// TIA Portal project "tiaS7libCommunication" (V15)

(* hardware
DEVICE "S7-1200 station_1"  S7-1200 Station
   slot 0: "Rack_0"  S7-1200 Rack  Rack  V1.0
   slot 1: "PLC_1"  CPU 1214C DC/DC/DC  6ES7 214-1AG40-0XB0  V4.2
DEVICE "HMI_1"  KTP700 Basic PN
   slot 0: "HMI_1"  KTP700 Basic PN  6AV2 123-2GB03-0AX0  15.0.0.0
   slot 1: "HMI_RT_1"  KTP700 Basic PN  6AV2 123-2GB03-0AX0  15.0.0.0
   slot 5: "HMI_1.IE_CP_1"  PROFINET Interface  15.0.0.0
      slot 1: "PROFINET Interface_1"  PROFINET Interface
         slot 1: "Port_1"  Port
DEVICE "HMI_2"  TP1500 Comfort
   slot 0: "HMI_2"  TP1500 Comfort  6AV2 124-0QC02-0AX1  15.0.0.0
   slot 1: "HMI_RT_2"  TP1500 Comfort  6AV2 124-0QC02-0AX1  15.0.0.0
   slot 5: "HMI_2.IE_CP_1"  PROFINET Interface  15.0.0.0
      slot 1: "PROFINET Interface_1"  PROFINET Interface
         slot 1: "Port_1"  Port
         slot 2: "Port_2"  Port
   slot 6: "HMI_2.IE_CP_2"  PROFINET Interface  15.0.0.0
      slot 1: "PROFINET Interface_GBit"  PROFINET Interface
         slot 1: "Port_1"  Port
   slot 7: "HMI_2.MPI/DP_CP_1"  MPI/DP Interface  15.0.0.0
*)

// ===== PLC "PLC_1"  CPU 1214C DC/DC/DC =====

VAR_GLOBAL   // PLC tag table "Default tag table"
   "o_test_valve_start" AT %M0.0 : Bool;
   "o_test_valve_end" AT %M0.1 : Bool;
   "i_test_valve_start" AT %M0.2 : Bool;
   "i_test_vavlve_end" AT %M0.3 : Bool;
END_VAR

TYPE "TestSuite"
   STRUCT
      tc_name : Array[1..64] of String[127];
      tc_size : Byte;
      ts_name : String[127];
   END_STRUCT;
END_TYPE

TYPE "UnitLib"
   STRUCT
      "step" : Int;
      input_buffer : Array[0..3] of Byte;
      output_buffer : Array[0..127] of Byte;
      output_len : UDInt;
      network_id : Conn_Ouc := 1;
      unit : Array[1..3] of "TestSuite";
      ts_size : Byte := 3;
   END_STRUCT;
   // unit[1].tc_size := 8;
   // unit[2].tc_name[2] := 'cb_insert_glass_test';
   // unit[2].tc_name[1] := 'cb_get_glass_info_test';
   // unit[1].ts_name := 'Priority queue test';
   // unit[2].tc_size := 16#7;
   // unit[1].tc_name[1] := 'pq_enqueue_test';
   // unit[1].tc_name[2] := 'pq_size_test';
   // unit[1].tc_name[3] := 'pq_is_empty_test';
   // unit[1].tc_name[8] := 'pq_clear_test';
   // unit[1].tc_name[4] := 'pq_peek_test';
   // unit[1].tc_name[5] := 'pq_delete_by_index_test';
   // unit[1].tc_name[6] := 'pq_dequeue_test';
   // unit[1].tc_name[7] := 'pq_find_by_vehicle_number_test';
   // unit[2].ts_name := 'Curing buffer test';
   // unit[2].tc_name[3] := 'cb_is_drawer_enabled_test';
   // unit[2].tc_name[4] := 'cb_is_drawer_free_test';
   // unit[2].tc_name[5] := 'cb_is_glass_expired_test';
   // unit[2].tc_name[7] := 'cb_remove_glass_test';
   // unit[2].tc_name[6] := 'cb_is_glass_ready_test';
   // unit[3].ts_name := 'Centering bed test';
   // unit[3].tc_name[1] := 'centering_bed_do_centering_test';
   // unit[3].tc_name[2] := 'centering_bed_get_state_test';
   // unit[3].tc_name[3] := 'centering_bed_is_centered_test';
   // unit[3].tc_name[4] := 'centering_bed_is_occupied_test';
   // unit[3].tc_name[5] := 'centering_bed_release_centering_test';
   // unit[3].tc_size := 16#5;
END_TYPE

TYPE "GlassInfo"
   STRUCT
      vehicle_number : String[100];
      vehicle_model : String[50];
      rear_window : String[50];
   END_STRUCT;
END_TYPE

TYPE "Valve2Pos"
   STRUCT
      status_error : Bool;   // error status, valve not reacts
      cmd_end_position : Bool;   // state conditional variable for setting valve end position
      cmd_start_position : Bool;   // state conditional variable for setting valve start position
      request_signal_start : Bool;   // request for set valve to start position
      request_signal_end : Bool;   // request for set valve to end position
      request_release : Bool;   // request for release valve (no output signals)
      watchdog_timer : TON_TIME;   // timer for reaction of valve
      reaction_delay : Time;   // delay for reaction of valve
      io : "IOValve2pos";
   END_STRUCT;
END_TYPE

// folder: CenteringBed

TYPE "CenteringBed"
   STRUCT
      "step" : Int;
      manual_mode_interface : "CenteringBedManual";
      x_centering_valve : "Valve2Pos";
      y_centering_valve : "Valve2Pos";
      suction_cup_lifting_cylinder : "Valve2Pos";
      status_error : Bool;
      cmd_vacuum : Bool;
      request_reset_error : Bool;
      io : "IOCenterngBed";
   END_STRUCT;
END_TYPE

TYPE "CenteringBedManual"
   STRUCT
      manual_mode : Bool;
      manual_anutomat_mode : Bool;
      request_manual_centering_x : Bool;
      request_manual_centering_y : Bool;
      request_manual_cuction_cup_lifting : Bool;
      request_manual_vacuum : Bool;
      request_manual_eject : Bool;
      request_do_manual_centering : Bool;
      request_manual_release_centering : Bool;
   END_STRUCT;
END_TYPE

// folder: CuringBuffer

TYPE "CuringBuffer"
   STRUCT
      drawer_array : Array[0..7] of "CuringBufferDrawer";
      min_expiration_time : Time;
      max_expiration_time : Time;
      drawer_count : Int := 8;
   END_STRUCT;
END_TYPE

TYPE "CuringBufferDrawer"
   STRUCT
      enable : Bool;
      occupied : Bool;
      presence_sensor : Bool;
      insertion_time : DTL;
      glass : "GlassInfo";
   END_STRUCT;
END_TYPE

// folder: MES

TYPE "MesPlcParams"
   STRUCT
      InitialPLC : Bool;   // InitialPLC
      InitialServerAck : Bool;   // InitialServerAck
      CycleRequest : Bool;   // CycleRequest
      CycleSuccess : Bool;   // CycleSuccess
      CycleFailure : Bool;   // CycleFailure
      CycleAbort : Bool;   // CycleAbort
      RES_501 : Byte;   // Reserviert
      RES_502 : Byte;   // Reserviert
      RES_503 : Byte;   // Reserviert
      PartSerialPLC : Array[1..40] of Char;   // PartSerialPLC
      ProcessDataCount : Int;   // ProcessDataCount <n>
      RES_546 : Array[0..126] of Word;   // Reserviert
      KeyProcessData : Array[1..50] of Char;   // Für jeden Index <i> von 0 bis <n> -1
      ValueProcessData : Array[1..50] of Char;   // Für jeden Index <i> von 0 bis <n> -1
   END_STRUCT;
   // PartSerialPLC[1] := '$00';
   // PartSerialPLC[2] := '$00';
   // PartSerialPLC[3] := '$00';
   // PartSerialPLC[4] := '$00';
   // PartSerialPLC[5] := '$00';
   // PartSerialPLC[6] := '$00';
   // PartSerialPLC[7] := '$00';
   // PartSerialPLC[8] := '$00';
   // PartSerialPLC[9] := '$00';
   // PartSerialPLC[10] := '$00';
   // PartSerialPLC[11] := '$00';
   // PartSerialPLC[12] := '$00';
   // PartSerialPLC[13] := '$00';
   // PartSerialPLC[14] := '$00';
   // PartSerialPLC[15] := '$00';
   // PartSerialPLC[16] := '$00';
   // PartSerialPLC[17] := '$00';
   // PartSerialPLC[18] := '$00';
   // PartSerialPLC[19] := '$00';
   // PartSerialPLC[20] := '$00';
   // PartSerialPLC[21] := '$00';
   // PartSerialPLC[22] := '$00';
   // PartSerialPLC[23] := '$00';
   // PartSerialPLC[24] := '$00';
   // PartSerialPLC[25] := '$00';
   // PartSerialPLC[26] := '$00';
   // PartSerialPLC[27] := '$00';
   // PartSerialPLC[28] := '$00';
   // PartSerialPLC[29] := '$00';
   // PartSerialPLC[30] := '$00';
   // PartSerialPLC[31] := '$00';
   // PartSerialPLC[32] := '$00';
   // PartSerialPLC[33] := '$00';
   // PartSerialPLC[34] := '$00';
   // PartSerialPLC[35] := '$00';
   // PartSerialPLC[36] := '$00';
   // PartSerialPLC[37] := '$00';
   // PartSerialPLC[38] := '$00';
   // PartSerialPLC[39] := '$00';
   // PartSerialPLC[40] := '$00';
   // KeyProcessData[1] := '$00';
   // KeyProcessData[2] := '$00';
   // KeyProcessData[3] := '$00';
   // KeyProcessData[4] := '$00';
   // KeyProcessData[5] := '$00';
   // KeyProcessData[6] := '$00';
   // KeyProcessData[7] := '$00';
   // KeyProcessData[8] := '$00';
   // KeyProcessData[9] := '$00';
   // KeyProcessData[10] := '$00';
   // KeyProcessData[11] := '$00';
   // KeyProcessData[12] := '$00';
   // KeyProcessData[13] := '$00';
   // KeyProcessData[14] := '$00';
   // KeyProcessData[15] := '$00';
   // KeyProcessData[16] := '$00';
   // KeyProcessData[17] := '$00';
   // KeyProcessData[18] := '$00';
   // KeyProcessData[19] := '$00';
   // KeyProcessData[20] := '$00';
   // KeyProcessData[21] := '$00';
   // KeyProcessData[22] := '$00';
   // KeyProcessData[23] := '$00';
   // KeyProcessData[24] := '$00';
   // KeyProcessData[25] := '$00';
   // KeyProcessData[26] := '$00';
   // KeyProcessData[27] := '$00';
   // KeyProcessData[28] := '$00';
   // KeyProcessData[29] := '$00';
   // KeyProcessData[30] := '$00';
   // KeyProcessData[31] := '$00';
   // KeyProcessData[32] := '$00';
   // KeyProcessData[33] := '$00';
   // KeyProcessData[34] := '$00';
   // KeyProcessData[35] := '$00';
   // KeyProcessData[36] := '$00';
   // KeyProcessData[37] := '$00';
   // KeyProcessData[38] := '$00';
   // KeyProcessData[39] := '$00';
   // KeyProcessData[40] := '$00';
   // KeyProcessData[41] := '$00';
   // KeyProcessData[42] := '$00';
   // KeyProcessData[43] := '$00';
   // KeyProcessData[44] := '$00';
   // KeyProcessData[45] := '$00';
   // KeyProcessData[46] := '$00';
   // KeyProcessData[47] := '$00';
   // KeyProcessData[48] := '$00';
   // KeyProcessData[49] := '$00';
   // KeyProcessData[50] := '$00';
   // ValueProcessData[1] := '$00';
   // ValueProcessData[2] := '$00';
   // ValueProcessData[3] := '$00';
   // ValueProcessData[4] := '$00';
   // ValueProcessData[5] := '$00';
   // ValueProcessData[6] := '$00';
   // ValueProcessData[7] := '$00';
   // ValueProcessData[8] := '$00';
   // ValueProcessData[9] := '$00';
   // ValueProcessData[10] := '$00';
   // ValueProcessData[11] := '$00';
   // ValueProcessData[12] := '$00';
   // ValueProcessData[13] := '$00';
   // ValueProcessData[14] := '$00';
   // ValueProcessData[15] := '$00';
   // ValueProcessData[16] := '$00';
   // ValueProcessData[17] := '$00';
   // ValueProcessData[18] := '$00';
   // ValueProcessData[19] := '$00';
   // ValueProcessData[20] := '$00';
   // ValueProcessData[21] := '$00';
   // ValueProcessData[22] := '$00';
   // ValueProcessData[23] := '$00';
   // ValueProcessData[24] := '$00';
   // ValueProcessData[25] := '$00';
   // ValueProcessData[26] := '$00';
   // ValueProcessData[27] := '$00';
   // ValueProcessData[28] := '$00';
   // ValueProcessData[29] := '$00';
   // ValueProcessData[30] := '$00';
   // ValueProcessData[31] := '$00';
   // ValueProcessData[32] := '$00';
   // ValueProcessData[33] := '$00';
   // ValueProcessData[34] := '$00';
   // ValueProcessData[35] := '$00';
   // ValueProcessData[36] := '$00';
   // ValueProcessData[37] := '$00';
   // ValueProcessData[38] := '$00';
   // ValueProcessData[39] := '$00';
   // ValueProcessData[40] := '$00';
   // ValueProcessData[41] := '$00';
   // ValueProcessData[42] := '$00';
   // ValueProcessData[43] := '$00';
   // ValueProcessData[44] := '$00';
   // ValueProcessData[45] := '$00';
   // ValueProcessData[46] := '$00';
   // ValueProcessData[47] := '$00';
   // ValueProcessData[48] := '$00';
   // ValueProcessData[49] := '$00';
   // ValueProcessData[50] := '$00';
END_TYPE

TYPE "MesServerParams"
   STRUCT
      LiveCheck : Bool;   // LiveCheck, vom Server gesetzt
      RES_001 : Byte;   // Reserviert
      InitialServer : Bool;   // InitialServer
      InitialPLCAck : Bool;   // InitialPLCAck
      ReadyForCycle : Bool;   // ReadyForCycle
      CycleRequestAck : Bool;   // CycleRequestAck
      CycleRequestReject : Bool;   // CycleRequestReject
      CycleAck : Bool;   // CycleAck
      RES_003 : Byte;   // Reserviert
      PartSerial : Array[1..40] of Char;   // PartSerial
      ParameterBarcode : Array[1..100] of Char;   // ParameterBarcode
      Error_Reason_Code : Int;
      ErrorMessage : Array[1..200] of Char;   // ErrorMessage
      Reserve : Array[1..154] of Char;   // Reserve
   END_STRUCT;
   // PartSerial[1] := '$00';
   // PartSerial[2] := '$00';
   // PartSerial[3] := '$00';
   // PartSerial[4] := '$00';
   // PartSerial[5] := '$00';
   // PartSerial[6] := '$00';
   // PartSerial[7] := '$00';
   // PartSerial[8] := '$00';
   // PartSerial[9] := '$00';
   // PartSerial[10] := '$00';
   // PartSerial[11] := '$00';
   // PartSerial[12] := '$00';
   // PartSerial[13] := '$00';
   // PartSerial[14] := '$00';
   // PartSerial[15] := '$00';
   // PartSerial[16] := '$00';
   // PartSerial[17] := '$00';
   // PartSerial[18] := '$00';
   // PartSerial[19] := '$00';
   // PartSerial[20] := '$00';
   // PartSerial[21] := '$00';
   // PartSerial[22] := '$00';
   // PartSerial[23] := '$00';
   // PartSerial[24] := '$00';
   // PartSerial[25] := '$00';
   // PartSerial[26] := '$00';
   // PartSerial[27] := '$00';
   // PartSerial[28] := '$00';
   // PartSerial[29] := '$00';
   // PartSerial[30] := '$00';
   // PartSerial[31] := '$00';
   // PartSerial[32] := '$00';
   // PartSerial[33] := '$00';
   // PartSerial[34] := '$00';
   // PartSerial[35] := '$00';
   // PartSerial[36] := '$00';
   // PartSerial[37] := '$00';
   // PartSerial[38] := '$00';
   // PartSerial[39] := '$00';
   // PartSerial[40] := '$00';
   // ParameterBarcode[1] := '$00';
   // ParameterBarcode[2] := '$00';
   // ParameterBarcode[3] := '$00';
   // ParameterBarcode[4] := '$00';
   // ParameterBarcode[5] := '$00';
   // ParameterBarcode[6] := '$00';
   // ParameterBarcode[7] := '$00';
   // ParameterBarcode[8] := '$00';
   // ParameterBarcode[9] := '$00';
   // ParameterBarcode[10] := '$00';
   // ParameterBarcode[11] := '$00';
   // ParameterBarcode[12] := '$00';
   // ParameterBarcode[13] := '$00';
   // ParameterBarcode[14] := '$00';
   // ParameterBarcode[15] := '$00';
   // ParameterBarcode[16] := '$00';
   // ParameterBarcode[17] := '$00';
   // ParameterBarcode[18] := '$00';
   // ParameterBarcode[19] := '$00';
   // ParameterBarcode[20] := '$00';
   // ParameterBarcode[21] := '$00';
   // ParameterBarcode[22] := '$00';
   // ParameterBarcode[23] := '$00';
   // ParameterBarcode[24] := '$00';
   // ParameterBarcode[25] := '$00';
   // ParameterBarcode[26] := '$00';
   // ParameterBarcode[27] := '$00';
   // ParameterBarcode[28] := '$00';
   // ParameterBarcode[29] := '$00';
   // ParameterBarcode[30] := '$00';
   // ParameterBarcode[31] := '$00';
   // ParameterBarcode[32] := '$00';
   // ParameterBarcode[33] := '$00';
   // ParameterBarcode[34] := '$00';
   // ParameterBarcode[35] := '$00';
   // ParameterBarcode[36] := '$00';
   // ParameterBarcode[37] := '$00';
   // ParameterBarcode[38] := '$00';
   // ParameterBarcode[39] := '$00';
   // ParameterBarcode[40] := '$00';
   // ParameterBarcode[41] := '$00';
   // ParameterBarcode[42] := '$00';
   // ParameterBarcode[43] := '$00';
   // ParameterBarcode[44] := '$00';
   // ParameterBarcode[45] := '$00';
   // ParameterBarcode[46] := '$00';
   // ParameterBarcode[47] := '$00';
   // ParameterBarcode[48] := '$00';
   // ParameterBarcode[49] := '$00';
   // ParameterBarcode[50] := '$00';
   // ParameterBarcode[51] := '$00';
   // ParameterBarcode[52] := '$00';
   // ParameterBarcode[53] := '$00';
   // ParameterBarcode[54] := '$00';
   // ParameterBarcode[55] := '$00';
   // ParameterBarcode[56] := '$00';
   // ParameterBarcode[57] := '$00';
   // ParameterBarcode[58] := '$00';
   // ParameterBarcode[59] := '$00';
   // ParameterBarcode[60] := '$00';
   // ParameterBarcode[61] := '$00';
   // ParameterBarcode[62] := '$00';
   // ParameterBarcode[63] := '$00';
   // ParameterBarcode[64] := '$00';
   // ParameterBarcode[65] := '$00';
   // ParameterBarcode[66] := '$00';
   // ParameterBarcode[67] := '$00';
   // ParameterBarcode[68] := '$00';
   // ParameterBarcode[69] := '$00';
   // ParameterBarcode[70] := '$00';
   // ParameterBarcode[71] := '$00';
   // ParameterBarcode[72] := '$00';
   // ParameterBarcode[73] := '$00';
   // ParameterBarcode[74] := '$00';
   // ParameterBarcode[75] := '$00';
   // ParameterBarcode[76] := '$00';
   // ParameterBarcode[77] := '$00';
   // ParameterBarcode[78] := '$00';
   // ParameterBarcode[79] := '$00';
   // ParameterBarcode[80] := '$00';
   // ParameterBarcode[81] := '$00';
   // ParameterBarcode[82] := '$00';
   // ParameterBarcode[83] := '$00';
   // ParameterBarcode[84] := '$00';
   // ParameterBarcode[85] := '$00';
   // ParameterBarcode[86] := '$00';
   // ParameterBarcode[87] := '$00';
   // ParameterBarcode[88] := '$00';
   // ParameterBarcode[89] := '$00';
   // ParameterBarcode[90] := '$00';
   // ParameterBarcode[91] := '$00';
   // ParameterBarcode[92] := '$00';
   // ParameterBarcode[93] := '$00';
   // ParameterBarcode[94] := '$00';
   // ParameterBarcode[95] := '$00';
   // ParameterBarcode[96] := '$00';
   // ParameterBarcode[97] := '$00';
   // ParameterBarcode[98] := '$00';
   // ParameterBarcode[99] := '$00';
   // ParameterBarcode[100] := '$00';
END_TYPE

// folder: PriorityQueue

TYPE "PriorityQueue"
   STRUCT
      array_size : Int := 100;
      size : Int;
      queue_array : Array[0..99] of "QueueNode";
   END_STRUCT;
END_TYPE

TYPE "QueueNode"
   STRUCT
      allocated : Bool;
      priority : Bool;
      glass : "GlassInfo";
   END_STRUCT;
END_TYPE

// folder: Queue

TYPE "queue_pc"
   STRUCT
      visual_queue : Array[0..9] of "GlassInfo";
      cmd_done : Bool;
   END_STRUCT;
END_TYPE

TYPE "queue_plc"
   STRUCT
      glass : "GlassInfo";
      cmd_add : Bool;
      cmd_add_priority : Bool;
      cmd_delete : Bool;
   END_STRUCT;
END_TYPE

// folder: io

TYPE "IOCuringBuffer"
   STRUCT
      presence_sensor_drawer_0 : Bool;
      presence_sensor_drawer_1 : Bool;
      presence_sensor_drawer_2 : Bool;
      presence_sensor_drawer_3 : Bool;
      presence_sensor_drawer_4 : Bool;
      presence_sensor_drawer_5 : Bool;
      presence_sensor_drawer_6 : Bool;
      presence_sensor_drawer_7 : Bool;
   END_STRUCT;
END_TYPE

TYPE "IOCenterngBed"
   STRUCT
      i_vacuum : Bool;
      i_glass_presence_sensor : Bool;
      o_vacuum : Bool;
      o_eject : Bool;
      centering_x_valve_io : "IOValve2pos";
      centering_y_valve_io : "IOValve2pos";
      suction_cup_lifting_io : "IOValve2pos";
   END_STRUCT;
END_TYPE

TYPE "IOValve2pos"
   STRUCT
      i_start_position : Bool;
      i_end_position : Bool;
      o_start_position : Bool;
      o_end_position : Bool;
   END_STRUCT;
END_TYPE

// folder: (top level)

DATA_BLOCK "PLCUnitLib_DB"   // DB2
{ S7_Optimized_Access := 'TRUE' }
VERSION : 0.1
// stored: InstanceOfName PLCUnitLib
"PLCUnitLib"
BEGIN
END_DATA_BLOCK

DATA_BLOCK "Valves_DB"   // DB3
{ S7_Optimized_Access := 'TRUE' }
VERSION : 0.1
   VAR
      test_valve : "Valve2Pos";
   END_VAR
BEGIN
END_DATA_BLOCK

DATA_BLOCK "io_sync_DB"   // DB4
{ S7_Optimized_Access := 'TRUE' }
VERSION : 0.1
// stored: InstanceOfName io_sync
"io_sync"
BEGIN
END_DATA_BLOCK

DATA_BLOCK "db_queue"   // DB5
{ S7_Optimized_Access := 'FALSE' }
VERSION : 0.1
   VAR
      plc : "queue_plc";
      pc : "queue_pc";
   END_VAR
BEGIN
   plc.glass.vehicle_number := '123456789 00';
   plc.glass.vehicle_model := 'IDBuzz';
   plc.glass.rear_window := 'VW-Number';
END_DATA_BLOCK

DATA_BLOCK "DB_MES_V2"   // DB6
{ S7_Optimized_Access := 'FALSE' }
VERSION : 0.1
   VAR
      MES : "MesServerParams";
      PLC : "MesPlcParams";
   END_VAR
BEGIN
END_DATA_BLOCK

DATA_BLOCK "DB_process_data"   // DB7
{ S7_Optimized_Access := 'TRUE' }
VERSION : 0.1
   VAR
      glass_queue : "PriorityQueue";
   END_VAR
   VAR RETAIN
      curing_buffer_1 : "CuringBuffer";
   END_VAR
   VAR
      centering_bed : "CenteringBed";
   END_VAR
BEGIN
END_DATA_BLOCK

DATA_BLOCK "DB_MES"   // DB600
{ S7_Optimized_Access := 'FALSE' }
VERSION : 0.1
   VAR
      LiveCheck : Bool;   // LiveCheck, vom Server gesetzt
      RES_001 : Byte;   // Reserviert
      InitialServer : Bool;   // InitialServer
      InitialPLCAck : Bool;   // InitialPLCAck
      ReadyForCycle : Bool;   // ReadyForCycle
      CycleRequestAck : Bool;   // CycleRequestAck
      CycleRequestReject : Bool;   // CycleRequestReject
      CycleAck : Bool;   // CycleAck
      RES_003 : Byte;   // Reserviert
      PartSerial : Array[1..40] of Char;   // PartSerial
      ParameterBarcode : Array[1..100] of Char;   // ParameterBarcode
      Error_Reason_Code : Int;
      ErrorMessage : Array[1..200] of Char;   // ErrorMessage
      Reserve : Array[1..154] of Char;   // Reserve
      InitialPLC : Bool;   // InitialPLC
      InitialServerAck : Bool;   // InitialServerAck
      CycleRequest : Bool;   // CycleRequest
      CycleSuccess : Bool;   // CycleSuccess
      CycleFailure : Bool;   // CycleFailure
      CycleAbort : Bool;   // CycleAbort
      RES_501 : Byte;   // Reserviert
      RES_502 : Byte;   // Reserviert
      RES_503 : Byte;   // Reserviert
      PartSerialPLC : Array[1..40] of Char;   // PartSerialPLC
      ProcessDataCount : Int;   // ProcessDataCount <n>
      RES_546 : Array[0..126] of Word;   // Reserviert
      KeyProcessData : Array[1..50] of Char;   // Für jeden Index <i> von 0 bis <n> -1
      ValueProcessData : Array[1..50] of Char;   // Für jeden Index <i> von 0 bis <n> -1
   END_VAR
BEGIN
   ValueProcessData[50] := '$00';
   ValueProcessData[1] := '$00';
   ValueProcessData[2] := '$00';
   ValueProcessData[3] := '$00';
   ValueProcessData[4] := '$00';
   ValueProcessData[5] := '$00';
   ValueProcessData[6] := '$00';
   ValueProcessData[7] := '$00';
   ValueProcessData[8] := '$00';
   ValueProcessData[9] := '$00';
   ValueProcessData[10] := '$00';
   ValueProcessData[11] := '$00';
   ValueProcessData[12] := '$00';
   ValueProcessData[13] := '$00';
   ValueProcessData[14] := '$00';
   ValueProcessData[15] := '$00';
   ValueProcessData[16] := '$00';
   ValueProcessData[17] := '$00';
   ValueProcessData[18] := '$00';
   ValueProcessData[19] := '$00';
   ValueProcessData[20] := '$00';
   ValueProcessData[21] := '$00';
   ValueProcessData[22] := '$00';
   ValueProcessData[23] := '$00';
   ValueProcessData[24] := '$00';
   ValueProcessData[25] := '$00';
   ValueProcessData[26] := '$00';
   ValueProcessData[27] := '$00';
   ValueProcessData[28] := '$00';
   ValueProcessData[29] := '$00';
   ValueProcessData[30] := '$00';
   ValueProcessData[31] := '$00';
   ValueProcessData[32] := '$00';
   ValueProcessData[33] := '$00';
   ValueProcessData[34] := '$00';
   ValueProcessData[35] := '$00';
   ValueProcessData[36] := '$00';
   ValueProcessData[37] := '$00';
   ValueProcessData[38] := '$00';
   ValueProcessData[39] := '$00';
   ValueProcessData[40] := '$00';
   ValueProcessData[41] := '$00';
   ValueProcessData[42] := '$00';
   ValueProcessData[43] := '$00';
   ValueProcessData[44] := '$00';
   ValueProcessData[45] := '$00';
   ValueProcessData[46] := '$00';
   ValueProcessData[47] := '$00';
   ValueProcessData[48] := '$00';
   ValueProcessData[49] := '$00';
   KeyProcessData[1] := '$00';
   KeyProcessData[2] := '$00';
   KeyProcessData[3] := '$00';
   KeyProcessData[4] := '$00';
   KeyProcessData[5] := '$00';
   KeyProcessData[6] := '$00';
   KeyProcessData[7] := '$00';
   KeyProcessData[8] := '$00';
   KeyProcessData[9] := '$00';
   KeyProcessData[10] := '$00';
   KeyProcessData[11] := '$00';
   KeyProcessData[12] := '$00';
   KeyProcessData[13] := '$00';
   KeyProcessData[14] := '$00';
   KeyProcessData[15] := '$00';
   KeyProcessData[16] := '$00';
   KeyProcessData[17] := '$00';
   KeyProcessData[18] := '$00';
   KeyProcessData[19] := '$00';
   KeyProcessData[20] := '$00';
   KeyProcessData[21] := '$00';
   KeyProcessData[22] := '$00';
   KeyProcessData[23] := '$00';
   KeyProcessData[24] := '$00';
   KeyProcessData[25] := '$00';
   KeyProcessData[26] := '$00';
   KeyProcessData[27] := '$00';
   KeyProcessData[28] := '$00';
   KeyProcessData[29] := '$00';
   KeyProcessData[30] := '$00';
   KeyProcessData[31] := '$00';
   KeyProcessData[32] := '$00';
   KeyProcessData[33] := '$00';
   KeyProcessData[34] := '$00';
   KeyProcessData[35] := '$00';
   KeyProcessData[36] := '$00';
   KeyProcessData[37] := '$00';
   KeyProcessData[38] := '$00';
   KeyProcessData[39] := '$00';
   KeyProcessData[40] := '$00';
   KeyProcessData[41] := '$00';
   KeyProcessData[42] := '$00';
   KeyProcessData[43] := '$00';
   KeyProcessData[44] := '$00';
   KeyProcessData[45] := '$00';
   KeyProcessData[46] := '$00';
   KeyProcessData[47] := '$00';
   KeyProcessData[48] := '$00';
   KeyProcessData[49] := '$00';
   KeyProcessData[50] := '$00';
   PartSerialPLC[1] := '$00';
   PartSerialPLC[2] := '$00';
   PartSerialPLC[3] := '$00';
   PartSerialPLC[4] := '$00';
   PartSerialPLC[5] := '$00';
   PartSerialPLC[6] := '$00';
   PartSerialPLC[7] := '$00';
   PartSerialPLC[8] := '$00';
   PartSerialPLC[9] := '$00';
   PartSerialPLC[10] := '$00';
   PartSerialPLC[11] := '$00';
   PartSerialPLC[12] := '$00';
   PartSerialPLC[13] := '$00';
   PartSerialPLC[14] := '$00';
   PartSerialPLC[15] := '$00';
   PartSerialPLC[16] := '$00';
   PartSerialPLC[17] := '$00';
   PartSerialPLC[18] := '$00';
   PartSerialPLC[19] := '$00';
   PartSerialPLC[20] := '$00';
   PartSerialPLC[21] := '$00';
   PartSerialPLC[22] := '$00';
   PartSerialPLC[23] := '$00';
   PartSerialPLC[24] := '$00';
   PartSerialPLC[25] := '$00';
   PartSerialPLC[26] := '$00';
   PartSerialPLC[27] := '$00';
   PartSerialPLC[28] := '$00';
   PartSerialPLC[29] := '$00';
   PartSerialPLC[30] := '$00';
   PartSerialPLC[31] := '$00';
   PartSerialPLC[32] := '$00';
   PartSerialPLC[33] := '$00';
   PartSerialPLC[34] := '$00';
   PartSerialPLC[35] := '$00';
   PartSerialPLC[36] := '$00';
   PartSerialPLC[37] := '$00';
   PartSerialPLC[38] := '$00';
   PartSerialPLC[39] := '$00';
   PartSerialPLC[40] := '$00';
   PartSerial[1] := '$00';
   PartSerial[2] := '$00';
   PartSerial[3] := '$00';
   PartSerial[4] := '$00';
   PartSerial[5] := '$00';
   PartSerial[6] := '$00';
   PartSerial[7] := '$00';
   PartSerial[8] := '$00';
   PartSerial[9] := '$00';
   PartSerial[10] := '$00';
   PartSerial[11] := '$00';
   PartSerial[12] := '$00';
   PartSerial[13] := '$00';
   PartSerial[14] := '$00';
   PartSerial[15] := '$00';
   PartSerial[16] := '$00';
   PartSerial[17] := '$00';
   PartSerial[18] := '$00';
   PartSerial[19] := '$00';
   PartSerial[20] := '$00';
   PartSerial[21] := '$00';
   PartSerial[22] := '$00';
   PartSerial[23] := '$00';
   PartSerial[24] := '$00';
   PartSerial[25] := '$00';
   PartSerial[26] := '$00';
   PartSerial[27] := '$00';
   PartSerial[28] := '$00';
   PartSerial[29] := '$00';
   PartSerial[30] := '$00';
   PartSerial[31] := '$00';
   PartSerial[32] := '$00';
   PartSerial[33] := '$00';
   PartSerial[34] := '$00';
   PartSerial[35] := '$00';
   PartSerial[36] := '$00';
   PartSerial[37] := '$00';
   PartSerial[38] := '$00';
   PartSerial[39] := '$00';
   PartSerial[40] := '$00';
   ParameterBarcode[1] := '$00';
   ParameterBarcode[2] := '$00';
   ParameterBarcode[3] := '$00';
   ParameterBarcode[4] := '$00';
   ParameterBarcode[5] := '$00';
   ParameterBarcode[6] := '$00';
   ParameterBarcode[7] := '$00';
   ParameterBarcode[8] := '$00';
   ParameterBarcode[9] := '$00';
   ParameterBarcode[10] := '$00';
   ParameterBarcode[11] := '$00';
   ParameterBarcode[12] := '$00';
   ParameterBarcode[13] := '$00';
   ParameterBarcode[14] := '$00';
   ParameterBarcode[15] := '$00';
   ParameterBarcode[16] := '$00';
   ParameterBarcode[17] := '$00';
   ParameterBarcode[18] := '$00';
   ParameterBarcode[19] := '$00';
   ParameterBarcode[20] := '$00';
   ParameterBarcode[21] := '$00';
   ParameterBarcode[22] := '$00';
   ParameterBarcode[23] := '$00';
   ParameterBarcode[24] := '$00';
   ParameterBarcode[25] := '$00';
   ParameterBarcode[26] := '$00';
   ParameterBarcode[27] := '$00';
   ParameterBarcode[28] := '$00';
   ParameterBarcode[29] := '$00';
   ParameterBarcode[30] := '$00';
   ParameterBarcode[31] := '$00';
   ParameterBarcode[32] := '$00';
   ParameterBarcode[33] := '$00';
   ParameterBarcode[34] := '$00';
   ParameterBarcode[35] := '$00';
   ParameterBarcode[36] := '$00';
   ParameterBarcode[37] := '$00';
   ParameterBarcode[38] := '$00';
   ParameterBarcode[39] := '$00';
   ParameterBarcode[40] := '$00';
   ParameterBarcode[41] := '$00';
   ParameterBarcode[42] := '$00';
   ParameterBarcode[43] := '$00';
   ParameterBarcode[44] := '$00';
   ParameterBarcode[45] := '$00';
   ParameterBarcode[46] := '$00';
   ParameterBarcode[47] := '$00';
   ParameterBarcode[48] := '$00';
   ParameterBarcode[49] := '$00';
   ParameterBarcode[50] := '$00';
   ParameterBarcode[51] := '$00';
   ParameterBarcode[52] := '$00';
   ParameterBarcode[53] := '$00';
   ParameterBarcode[54] := '$00';
   ParameterBarcode[55] := '$00';
   ParameterBarcode[56] := '$00';
   ParameterBarcode[57] := '$00';
   ParameterBarcode[58] := '$00';
   ParameterBarcode[59] := '$00';
   ParameterBarcode[60] := '$00';
   ParameterBarcode[61] := '$00';
   ParameterBarcode[62] := '$00';
   ParameterBarcode[63] := '$00';
   ParameterBarcode[64] := '$00';
   ParameterBarcode[65] := '$00';
   ParameterBarcode[66] := '$00';
   ParameterBarcode[67] := '$00';
   ParameterBarcode[68] := '$00';
   ParameterBarcode[69] := '$00';
   ParameterBarcode[70] := '$00';
   ParameterBarcode[71] := '$00';
   ParameterBarcode[72] := '$00';
   ParameterBarcode[73] := '$00';
   ParameterBarcode[74] := '$00';
   ParameterBarcode[75] := '$00';
   ParameterBarcode[76] := '$00';
   ParameterBarcode[77] := '$00';
   ParameterBarcode[78] := '$00';
   ParameterBarcode[79] := '$00';
   ParameterBarcode[80] := '$00';
   ParameterBarcode[81] := '$00';
   ParameterBarcode[82] := '$00';
   ParameterBarcode[83] := '$00';
   ParameterBarcode[84] := '$00';
   ParameterBarcode[85] := '$00';
   ParameterBarcode[86] := '$00';
   ParameterBarcode[87] := '$00';
   ParameterBarcode[88] := '$00';
   ParameterBarcode[89] := '$00';
   ParameterBarcode[90] := '$00';
   ParameterBarcode[91] := '$00';
   ParameterBarcode[92] := '$00';
   ParameterBarcode[93] := '$00';
   ParameterBarcode[94] := '$00';
   ParameterBarcode[95] := '$00';
   ParameterBarcode[96] := '$00';
   ParameterBarcode[97] := '$00';
   ParameterBarcode[98] := '$00';
   ParameterBarcode[99] := '$00';
   ParameterBarcode[100] := '$00';
END_DATA_BLOCK

// folder: unitLib

DATA_BLOCK "PLC_1_Connection_DB"   // DB1
{ S7_Optimized_Access := 'TRUE' }
AUTHOR : SIMATIC
FAMILY : MC7Plus
NAME : TC_IP_v4
VERSION : 1.0
// stored: InstanceOfName TCON_IP_v4
"TCON_IP_v4"
BEGIN
   ID := 1;
   InterfaceId := 64;
   LocalPort := 2500;
END_DATA_BLOCK

// folder: (top level)

FUNCTION "pc_queue_runtime" : Void   // FC73, SCL
{ S7_Optimized_Access := 'TRUE' }
VERSION : 0.1
BEGIN

   IF "db_queue".plc.cmd_add_priority = TRUE
       OR "db_queue".plc.cmd_add = true
       OR "db_queue".plc.cmd_delete = TRUE

   THEN
       IF "db_queue".pc.cmd_done = TRUE
       THEN
           "db_queue".plc.cmd_add_priority := false;
           "db_queue".plc.cmd_add := false;
           "db_queue".plc.cmd_delete := false;
           "db_queue".pc.cmd_done := false;
       END_IF;
   END_IF;
END_FUNCTION

ORGANIZATION_BLOCK "Main"   // OB1, LAD, ProgramCycle
TITLE = "Main Program Sweep (Cycle)"
{ S7_Optimized_Access := 'TRUE' }
VERSION : 0.1
   VAR_INPUT
      Initial_Call : Bool;   // Initial call of this OB
      Remanence : Bool;   // =True, if remanent data are available
   END_VAR
   VAR_TEMP
      ret_value : Bool;
   END_VAR
BEGIN

REGION Network 1
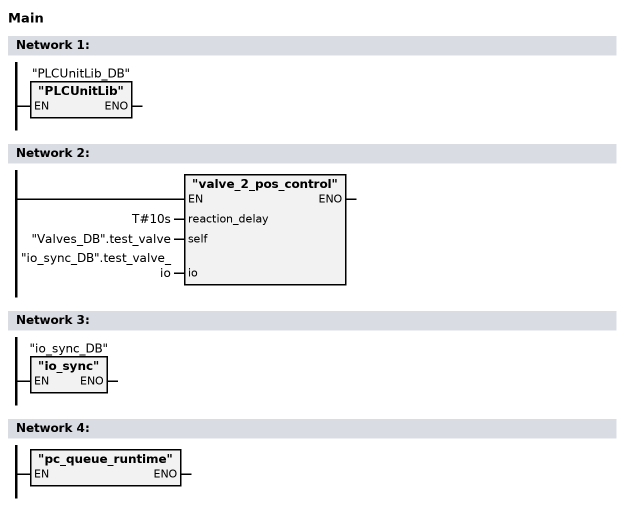
   RUNG wire#powerrail
      "PLCUnitLib_DB"()
   END_RUNG
   // the same network as SCL:
   "PLCUnitLib_DB"();   // "PLCUnitLib"
END_REGION

REGION Network 2
   RUNG wire#powerrail
      "valve_2_pos_control"(reaction_delay := T#10s, self := "Valves_DB".test_valve, io := "io_sync_DB".test_valve_io)
   END_RUNG
   // the same network as SCL:
   "valve_2_pos_control"(reaction_delay := T#10s,
                         self := "Valves_DB".test_valve,
                         io := "io_sync_DB".test_valve_io);
END_REGION

REGION Network 3
   RUNG wire#powerrail
      "io_sync_DB"()
   END_RUNG
   // the same network as SCL:
   "io_sync_DB"();   // "io_sync"
END_REGION

REGION Network 4
   RUNG wire#powerrail
      "pc_queue_runtime"()
   END_RUNG
   // the same network as SCL:
   "pc_queue_runtime"();
END_REGION
END_ORGANIZATION_BLOCK

// folder: CenteringBed

FUNCTION "centering_bed_runtime" : Void   // FC53, SCL
{ S7_Optimized_Access := 'TRUE' }
VERSION : 0.1
   VAR_INPUT
      valve_reaction_delay : Time;   // retain settings
   END_VAR
   VAR_IN_OUT
      self : "CenteringBed";
      io : "IOCenterngBed";
   END_VAR
BEGIN



   "centering_station_valve_control"(valve_reaction_delay:=#valve_reaction_delay, self:=#self);
   "centering_bed_manual_mod_control"(self := #self);
   "centering_bed_stepper"(self:=#self);
   "centering_bed_catch_error"(self:=#self);
END_FUNCTION

// folder: CenteringBed/api

FUNCTION "centering_bed_is_centered" : Bool   // FC54, SCL
{ S7_Optimized_Access := 'TRUE' }
VERSION : 0.1
   VAR_IN_OUT
      self : "CenteringBed";
   END_VAR
BEGIN


   #centering_bed_is_centered := false;
END_FUNCTION

FUNCTION "centering_bed_do_centering" : Bool   // FC55, SCL
{ S7_Optimized_Access := 'TRUE' }
VERSION : 0.1
   VAR_IN_OUT
      self : "CenteringBed";
   END_VAR
BEGIN



   #centering_bed_do_centering := false;
END_FUNCTION

FUNCTION "centering_bed_is_occupied" : Bool   // FC56, SCL
{ S7_Optimized_Access := 'TRUE' }
VERSION : 0.1
   VAR_IN_OUT
      self : "CenteringBed";
   END_VAR
BEGIN


   #centering_bed_is_occupied := false;
END_FUNCTION

FUNCTION "centering_bed_get_state" : Bool   // FC57, SCL
{ S7_Optimized_Access := 'TRUE' }
VERSION : 0.1
   VAR_IN_OUT
      self : "CenteringBed";
   END_VAR
BEGIN



   #centering_bed_get_state := false;
END_FUNCTION

FUNCTION "centering_bed_release_centering" : Bool   // FC58, SCL
{ S7_Optimized_Access := 'TRUE' }
VERSION : 0.1
   VAR_IN_OUT
      self : "CenteringBed";
   END_VAR
BEGIN


   #centering_bed_release_centering := false;
END_FUNCTION

// folder: CenteringBed/fce

FUNCTION "centering_bed_stepper" : Void   // FC66, SCL
{ S7_Optimized_Access := 'TRUE' }
VERSION : 0.1
   VAR_IN_OUT
      self : "CenteringBed";
   END_VAR
   VAR CONSTANT
      STEP_RELEASE : Int := 0;
      STEP_CENTERING_CHECK_GLASS_PRESENCE : Int := 1;
      STEP_CENTERING_Y : Int := 2;
      STEP_CENTERING_X : Int := 3;
      STEP_CENTERING_SUCTION_CUP_LIFING_UP : Int := 4;
      STEP_CENTERING_VACUUM_ON : Int := 5;
      STEP_RELEASE_CENTERING : Int := 6;
      STEP_CENTERED : Int := 7;
      STEP_RELEASING_VACUUM_OFF : Int := 8;
      STEP_RELEASING_SUCTION_CUP_LIFTING_DOWN : Int := 9;
      STEP_RESET : Int := 10;
      STEP_ERROR : Int := 128;
   END_VAR
BEGIN



   IF #self.step = #STEP_CENTERING_VACUUM_ON
       OR #self.step = #STEP_CENTERED
       OR #self.step = #STEP_RELEASE_CENTERING
   THEN
       #self.cmd_vacuum := true;
   ELSE
       #self.cmd_vacuum := false;
   END_IF;

   #self.suction_cup_lifting_cylinder.request_release := #self.step >= #STEP_ERROR;
   #self.x_centering_valve.request_release := #self.step >= #STEP_ERROR;
   #self.y_centering_valve.request_release := #self.step >= #STEP_ERROR;


   (*
   ** glass must be present during centering
   *)


   IF #self.manual_mode_interface.manual_mode = false
       AND #self.step > #STEP_RELEASE
       AND #self.step <= #STEP_CENTERED
       AND #self.io.i_glass_presence_sensor = FALSE
   THEN
       #self.step := #STEP_ERROR;
   END_IF;



   CASE #self.step OF
       #STEP_RELEASE:
           ;

       #STEP_CENTERED:
           ;

       #STEP_CENTERING_CHECK_GLASS_PRESENCE:
           IF #self.io.i_glass_presence_sensor = TRUE
               OR #self.manual_mode_interface.manual_mode = true
           THEN
               #self.step := #STEP_CENTERING_Y;
           ELSE
               #self.step := #STEP_ERROR;
           END_IF;

       #STEP_CENTERING_Y:
           "valve_2_pos_set_end_position"(#self.y_centering_valve);

           IF "valve_2_pos_is_end_position"(#self.y_centering_valve) = true
           THEN
               #self.step := #STEP_CENTERING_X;
           END_IF;

       #STEP_CENTERING_X:
           "valve_2_pos_set_end_position"(#self.x_centering_valve);

           IF "valve_2_pos_is_end_position"(#self.x_centering_valve) = true
           THEN
               #self.step := #STEP_CENTERING_SUCTION_CUP_LIFING_UP;
           END_IF;

       #STEP_CENTERING_SUCTION_CUP_LIFING_UP:
           "valve_2_pos_set_end_position"(#self.suction_cup_lifting_cylinder);

           IF "valve_2_pos_is_end_position"(#self.suction_cup_lifting_cylinder) = true
           THEN
               #self.step := #STEP_CENTERING_VACUUM_ON;
           END_IF;

       #STEP_CENTERING_VACUUM_ON:
           IF #self.io.i_vacuum = TRUE
           THEN
               #self.step := #STEP_RELEASE_CENTERING;
           END_IF;

       #STEP_RELEASE_CENTERING:
           "valve_2_pos_set_start_position"(#self.y_centering_valve);
           "valve_2_pos_set_start_position"(#self.x_centering_valve);

           IF "valve_2_pos_is_start_position"(#self.y_centering_valve) = TRUE
               AND "valve_2_pos_is_start_position"(#self.x_centering_valve) = TRUE
           THEN
               #self.step := #STEP_CENTERED;
           END_IF;

       #STEP_RELEASING_VACUUM_OFF:
           #self.io.o_eject := #self.io.i_vacuum;

           IF #self.io.i_vacuum = false
           THEN
               #self.step := #STEP_RELEASING_SUCTION_CUP_LIFTING_DOWN;
           END_IF;

       #STEP_RELEASING_SUCTION_CUP_LIFTING_DOWN:
           "valve_2_pos_set_start_position"(#self.suction_cup_lifting_cylinder);

           IF "valve_2_pos_is_start_position"(#self.suction_cup_lifting_cylinder) = TRUE
           THEN
               #self.step := #STEP_RELEASE;
           END_IF;
       #STEP_RESET:
           #self.io.o_eject := #self.io.i_vacuum;

           IF #self.io.i_vacuum = false
           THEN
               "valve_2_pos_set_start_position"(#self.suction_cup_lifting_cylinder);
               "valve_2_pos_set_start_position"(#self.y_centering_valve);
               "valve_2_pos_set_start_position"(#self.x_centering_valve);

               IF "valve_2_pos_is_start_position"(#self.suction_cup_lifting_cylinder) = TRUE
                   AND "valve_2_pos_is_start_position"(#self.y_centering_valve) = TRUE
                   AND "valve_2_pos_is_start_position"(#self.x_centering_valve) = TRUE
               THEN
                   #self.step := #STEP_RELEASE;
               END_IF;
           END_IF;
       ELSE
           #self.step := #STEP_ERROR;
   END_CASE;
END_FUNCTION

FUNCTION "centering_station_valve_control" : Void   // FC67, SCL
{ S7_Optimized_Access := 'TRUE' }
VERSION : 0.1
   VAR_INPUT
      valve_reaction_delay : Time;
   END_VAR
   VAR_IN_OUT
      self : "CenteringBed";
   END_VAR
BEGIN



   (*
   ** control of x centering valve
   *)
   "valve_2_pos_control"(self := #self.x_centering_valve,
                   io:=#self.io.centering_x_valve_io,
                   reaction_delay := #valve_reaction_delay);

   (*
   ** control of y centering valve
   *) 
   "valve_2_pos_control"(self := #self.y_centering_valve,
                   io:=#self.io.centering_y_valve_io,
                   reaction_delay := #valve_reaction_delay);

   (*
   ** control of suction cup lifting valve
   *)
   "valve_2_pos_control"(self := #self.suction_cup_lifting_cylinder,
                   io:=#self.io.suction_cup_lifting_io,
                   reaction_delay := #valve_reaction_delay);
END_FUNCTION

FUNCTION "centering_bed_catch_error" : Void   // FC68, LAD
{ S7_Optimized_Access := 'TRUE' }
VERSION : 0.1
   VAR_IN_OUT
      self : "CenteringBed";
   END_VAR
BEGIN

REGION Network 1: catch error
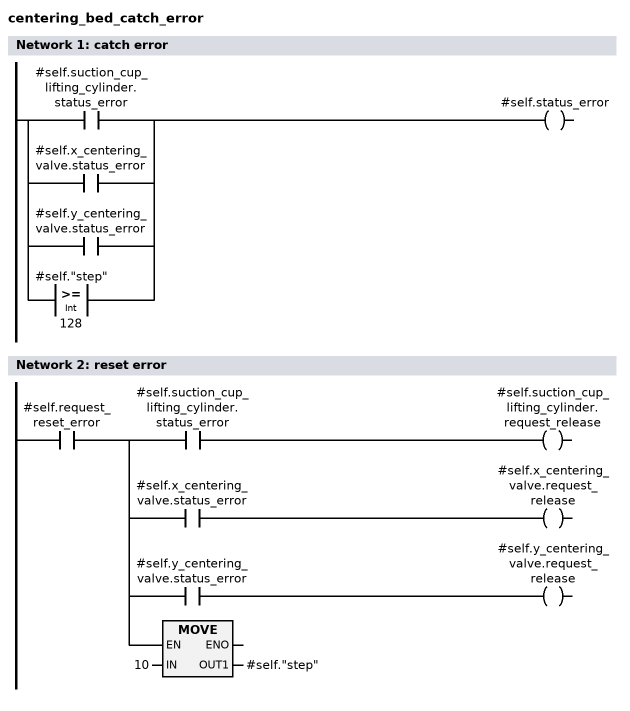
   RUNG wire#powerrail
      Contact( #self.suction_cup_lifting_cylinder.status_error )
      wire#w1
      Coil( #self.status_error )
   END_RUNG
   RUNG wire#powerrail
      Contact( #self.x_centering_valve.status_error )
   END_RUNG wire#w1
   RUNG wire#powerrail
      Contact( #self.y_centering_valve.status_error )
   END_RUNG wire#w1
   RUNG wire#powerrail
      { S7_Templates := "SrcType := Int" } GE_Contact(in1 := #self."step", in2 := 128)
   END_RUNG wire#w1
   // the same network as SCL:
   #self.status_error := #self.suction_cup_lifting_cylinder.status_error OR #self.x_centering_valve.status_error OR #self.y_centering_valve.status_error OR (#self."step" >= 128);
END_REGION

REGION Network 2: reset error
   RUNG wire#powerrail
      Contact( #self.request_reset_error )
      wire#w1
      Contact( #self.suction_cup_lifting_cylinder.status_error )
      Coil( #self.suction_cup_lifting_cylinder.request_release )
   END_RUNG
   RUNG wire#w1
      Contact( #self.x_centering_valve.status_error )
      Coil( #self.x_centering_valve.request_release )
   END_RUNG
   RUNG wire#w1
      Contact( #self.y_centering_valve.status_error )
      Coil( #self.y_centering_valve.request_release )
   END_RUNG
   RUNG wire#w1
      Move(in := 10, out1 => #self."step")
   END_RUNG
   // the same network as SCL:
   #self.suction_cup_lifting_cylinder.request_release := #self.request_reset_error AND #self.suction_cup_lifting_cylinder.status_error;
   #self.x_centering_valve.request_release := #self.request_reset_error AND #self.x_centering_valve.status_error;
   #self.y_centering_valve.request_release := #self.request_reset_error AND #self.y_centering_valve.status_error;
   IF #self.request_reset_error THEN #self."step" := 10; END_IF;
END_REGION
END_FUNCTION

FUNCTION "centering_bed_manual_mod_control" : Void   // FC71, SCL
{ S7_Optimized_Access := 'TRUE' }
VERSION : 0.1
   VAR_IN_OUT
      self : "CenteringBed";
   END_VAR
BEGIN
END_FUNCTION

// folder: CuringBuffer

FUNCTION "cb_runtime" : Void   // FC44, SCL
{ S7_Optimized_Access := 'TRUE' }
VERSION : 0.1
// Synchronize input signals from presence sensor inside drawers with data structure
   VAR_INPUT
      min_expiration_time : Time;
      max_expiration_time : Time;
      io : "IOCuringBuffer";
   END_VAR
   VAR_IN_OUT
      self : "CuringBuffer";
   END_VAR
BEGIN
   #self.min_expiration_time := #min_expiration_time;
   #self.max_expiration_time := #max_expiration_time;

   #self.drawer_array[0].presence_sensor := #io.presence_sensor_drawer_0;
   #self.drawer_array[1].presence_sensor := #io.presence_sensor_drawer_1;
   #self.drawer_array[2].presence_sensor := #io.presence_sensor_drawer_2;
   #self.drawer_array[3].presence_sensor := #io.presence_sensor_drawer_3;
   #self.drawer_array[4].presence_sensor := #io.presence_sensor_drawer_4;
   #self.drawer_array[5].presence_sensor := #io.presence_sensor_drawer_5;
   #self.drawer_array[6].presence_sensor := #io.presence_sensor_drawer_6;
   #self.drawer_array[7].presence_sensor := #io.presence_sensor_drawer_7;
END_FUNCTION

// folder: CuringBuffer/api

FUNCTION "cb_insert_glass" : Bool   // FC32, SCL
{ S7_Optimized_Access := 'TRUE' }
VERSION : 0.1
   VAR_INPUT
      drawer_index : Int;
      glass : "GlassInfo";
   END_VAR
   VAR_IN_OUT
      self : "CuringBuffer";
   END_VAR
   VAR_TEMP
      ret_value : Int;
   END_VAR
BEGIN

   IF #drawer_index < #self.drawer_count
       AND #self.drawer_array[#drawer_index].enable = TRUE
       AND #self.drawer_array[#drawer_index].occupied = false
   THEN
       #ret_value := RD_SYS_T(#self.drawer_array[#drawer_index].insertion_time);
       #self.drawer_array[#drawer_index].glass := #glass;
       #self.drawer_array[#drawer_index].occupied := true;

       #cb_insert_glass := true;
   ELSE
       #cb_insert_glass := false;
   END_IF;
END_FUNCTION

FUNCTION "cb_is_drawer_free" : Bool   // FC33, SCL
{ S7_Optimized_Access := 'TRUE' }
VERSION : 0.1
   VAR_INPUT
      drawer_index : Int;
   END_VAR
   VAR_IN_OUT
      self : "CuringBuffer";
   END_VAR
BEGIN

   IF #drawer_index < #self.drawer_count
       AND #self.drawer_array[#drawer_index].enable = TRUE
       AND #self.drawer_array[#drawer_index].occupied = FALSE
       AND #self.drawer_array[#drawer_index].presence_sensor = false
   THEN
       #cb_is_drawer_free := true;
   ELSE
       #cb_is_drawer_free := false;
   END_IF;
END_FUNCTION

FUNCTION "cb_is_drawer_enabled" : Bool   // FC34, SCL
{ S7_Optimized_Access := 'TRUE' }
VERSION : 0.1
   VAR_INPUT
      drawer_index : Int;
   END_VAR
   VAR_IN_OUT
      self : "CuringBuffer";
   END_VAR
BEGIN

   IF #drawer_index < #self.drawer_count
       AND #self.drawer_array[#drawer_index].enable = TRUE
   THEN
       #cb_is_drawer_enabled := true;
   ELSE
       #cb_is_drawer_enabled := false;
   END_IF;
END_FUNCTION

FUNCTION "cb_remove_glass" : Bool   // FC35, SCL
{ S7_Optimized_Access := 'TRUE' }
VERSION : 0.1
   VAR_INPUT
      drawer_index : Int;
   END_VAR
   VAR_IN_OUT
      self : "CuringBuffer";
   END_VAR
BEGIN
   IF "cb_is_drawer_free"(drawer_index := #drawer_index, self := #self) = false
   THEN
       #self.drawer_array[#drawer_index].occupied := false;
       #cb_remove_glass := true;
   ELSE
       #cb_remove_glass := false;
   END_IF;
END_FUNCTION

FUNCTION "cb_is_glass_expired" : Bool   // FC36, SCL
{ S7_Optimized_Access := 'TRUE' }
VERSION : 0.1
   VAR_INPUT
      drawer_index : Int;
   END_VAR
   VAR_IN_OUT
      self : "CuringBuffer";
   END_VAR
   VAR_TEMP
      current_time : DTL;
      ret_value : Int;
      time_difference : Time;
   END_VAR
BEGIN

   IF "cb_is_drawer_enabled"(drawer_index := #drawer_index, self := #self) = true
       AND "cb_is_drawer_free"(drawer_index := #drawer_index, self := #self) = FALSE
   THEN
       #ret_value := RD_SYS_T(#current_time);
       #time_difference := T_DIFF(IN1 := #current_time, IN2 := #self.drawer_array[#drawer_index].insertion_time);

       IF #time_difference <= #self.max_expiration_time
       THEN
           #cb_is_glass_expired := true;
       ELSE
           #cb_is_glass_expired := false;
       END_IF;
   ELSE
       #cb_is_glass_expired := false;
   END_IF;
END_FUNCTION

FUNCTION "cb_get_class_info" : "GlassInfo"   // FC37, SCL
{ S7_Optimized_Access := 'TRUE' }
VERSION : 0.1
   VAR_INPUT
      drawer_index : Int;
   END_VAR
   VAR_IN_OUT
      self : "CuringBuffer";
   END_VAR
   VAR_TEMP
      glass : "GlassInfo";
   END_VAR
BEGIN

   IF #drawer_index < #self.drawer_count
       AND #self.drawer_array[#drawer_index].enable = true
       AND #self.drawer_array[#drawer_index].occupied = TRUE
   THEN
       #glass := #self.drawer_array[#drawer_index].glass;
   END_IF;

   #cb_get_class_info := #glass;
END_FUNCTION

FUNCTION "cb_is_glass_ready" : Bool   // FC47, SCL
{ S7_Optimized_Access := 'TRUE' }
VERSION : 0.1
   VAR_INPUT
      drawer_index : Int;
   END_VAR
   VAR_IN_OUT
      self : "CuringBuffer";
   END_VAR
   VAR_TEMP
      current_time : DTL;
      ret_value : Int;
      time_difference : Time;
   END_VAR
BEGIN


   IF  "cb_is_drawer_enabled"(drawer_index := #drawer_index, self := #self) = true
       AND "cb_is_drawer_free"(drawer_index := #drawer_index, self := #self) = FALSE
   THEN
       #ret_value := RD_SYS_T(#current_time);
       #time_difference := T_DIFF(IN1 := #current_time, IN2 := #self.drawer_array[#drawer_index].insertion_time);

       IF #self.min_expiration_time <= #time_difference
       THEN
           #cb_is_glass_ready := true;
       ELSE
           #cb_is_glass_ready := false;
       END_IF;
   ELSE
       #cb_is_glass_ready := false;
   END_IF;
END_FUNCTION

// folder: GlassInfo

FUNCTION "gi_new" : "GlassInfo"   // FC27, SCL
{ S7_Optimized_Access := 'TRUE' }
VERSION : 0.1
// Initialize the glass_info structure and return it as result for next use
   VAR_INPUT
      rear_window : String;
      vehicle_model : String;
      vehicle_number : String;
   END_VAR
   VAR_TEMP
      glass : "GlassInfo";
   END_VAR
BEGIN


   #glass.rear_window := #rear_window;
   #glass.vehicle_number := #vehicle_number;
   #glass.vehicle_model := #vehicle_model;

   #gi_new := #glass;
END_FUNCTION

FUNCTION "gi_compare_vehicle_numbers" : Bool   // FC29, SCL
{ S7_Optimized_Access := 'TRUE' }
VERSION : 0.1
// Compares two vehicle numbers except rework indexes and return true value if are the same glass
   VAR_INPUT
      vehicle_number_1 : String;
      vehicle_number_2 : String;
   END_VAR
   VAR_TEMP
      vn_1_length : Int;
      vn_2_length : Int;
   END_VAR
BEGIN

   (*
   ** compare two vehicle numbers except revork index
   *)

   #vn_1_length := FIND(IN1 := #vehicle_number_1, IN2 := ' ');
   #vn_2_length := FIND(IN1 := #vehicle_number_2, IN2 := ' ');

   IF LEFT(IN := #vehicle_number_1, L := #vn_1_length) = LEFT(IN := #vehicle_number_2, L := #vn_2_length)
   THEN
       #gi_compare_vehicle_numbers := true;
   ELSE
       #gi_compare_vehicle_numbers := false;
   END_IF;
END_FUNCTION

// folder: PriorityQueue

FUNCTION "pq_enqueue" : Bool   // FC11, SCL
{ S7_Optimized_Access := 'TRUE' }
VERSION : 0.1
// Inserts new data to last array item in order, or updates glass parameters if  the vehicle number is already in queue
   VAR_INPUT
      glass : "GlassInfo";
      priority : Bool;
   END_VAR
   VAR_IN_OUT
      self : "PriorityQueue";
   END_VAR
   VAR_TEMP
      node_index : Int;
   END_VAR
BEGIN

   IF #self.size < #self.array_size
   THEN
       #node_index := "pq_find_by_vehicle_number"(vehicle_number := #glass.vehicle_number, self := #self);

       IF #node_index < 0
       THEN
           IF #priority = TRUE
           THEN
               "pg_shift_right"(#self);

               #self.queue_array[0].glass := #glass;
               #self.queue_array[0].priority := true;
               #self.queue_array[0].allocated := true;
           ELSE
               #self.queue_array[#self.size].glass := #glass;
               #self.queue_array[#self.size].allocated := true;
               #self.queue_array[0].priority := false;
           END_IF;

           #self.size := #self.size + 1;
       ELSE
           #self.queue_array[#node_index].glass := #glass;
       END_IF;

       #pq_enqueue := true;
   ELSE
       #pq_enqueue := false;
   END_IF;
END_FUNCTION

FUNCTION "pq_dequeue" : Bool   // FC12, SCL
{ S7_Optimized_Access := 'TRUE' }
VERSION : 0.1
// Deletes the firest array item in order and shift all next data to left and initialize the last item in order
   VAR_IN_OUT
      self : "PriorityQueue";
   END_VAR
BEGIN

   IF "pq_size"(#self) > 0
   THEN
       IF "pq_size"(#self) >= 2
       THEN
           "pg_shift_left"(#self);
       END_IF;

       #self.queue_array[#self.size - 1].allocated := false;
       #self.queue_array[#self.size - 1].priority := false;
       #self.size := #self.size - 1;

       #pq_dequeue := true;
   ELSE
       #pq_dequeue := false;
   END_IF;
END_FUNCTION

FUNCTION "pq_peek" : "QueueNode"   // FC13, SCL
{ S7_Optimized_Access := 'TRUE' }
VERSION : 0.1
// Return glass_info structure with glass parameters on given position in queue (array), or return empty glass_info structure if index is out of range
   VAR_INPUT
      index : Int;
   END_VAR
   VAR_IN_OUT
      self : "PriorityQueue";
   END_VAR
   VAR_TEMP
      node : "QueueNode";
   END_VAR
BEGIN

   IF #index < "pq_size"(#self)
   THEN
       #node := #self.queue_array[#index];
   END_IF;

   #pq_peek := #node;
END_FUNCTION

FUNCTION "pq_delete_by_index" : Bool   // FC14, SCL
{ S7_Optimized_Access := 'TRUE' }
VERSION : 0.2
// Deletes data from array and shift all next data one position to left, and initialize last array item in order
   VAR_INPUT
      index : Int;
   END_VAR
   VAR_IN_OUT
      self : "PriorityQueue";
   END_VAR
   VAR_TEMP
      i : Int;
   END_VAR
BEGIN

   IF #index < "pq_size"(#self)
   THEN
       #i := #index;

       WHILE #i < "pq_size"(#self)-1 DO
           #self.queue_array[#i] := #self.queue_array[#i + 1];
           #i := #i + 1;
       END_WHILE;

       #self.queue_array[#self.size - 1].allocated := false;
       #self.queue_array[#self.size - 1].priority := false;
       #self.size := #self.size - 1;

       #pq_delete_by_index := true;
   ELSE
       #pq_delete_by_index := false;
   END_IF;
END_FUNCTION

FUNCTION "pq_is_empty" : Bool   // FC15, SCL
{ S7_Optimized_Access := 'TRUE' }
VERSION : 0.1
// Check if the queue is empty or not
   VAR_IN_OUT
      self : "PriorityQueue";
   END_VAR
BEGIN

   IF #self.size > 0
   THEN
       #pq_is_empty := false;
   ELSE
       #pq_is_empty := true;
   END_IF;
END_FUNCTION

FUNCTION "pq_size" : Int   // FC16, SCL
{ S7_Optimized_Access := 'TRUE' }
VERSION : 0.1
// Return number of allocated items in queue
   VAR_IN_OUT
      self : "PriorityQueue";
   END_VAR
BEGIN


   #pq_size := #self.size;
END_FUNCTION

FUNCTION "pq_find_by_vehicle_number" : Int   // FC18, SCL
{ S7_Optimized_Access := 'TRUE' }
VERSION : 0.1
// Fineds and return the position of array item where is glass with given vehicle number, or return -1 value if the glass with given vehicle number is not inside
   VAR_INPUT
      vehicle_number : String;
   END_VAR
   VAR_IN_OUT
      self : "PriorityQueue";
   END_VAR
   VAR_TEMP
      i : Int;
   END_VAR
BEGIN

   #pq_find_by_vehicle_number := -1;

   IF "pq_is_empty"(#self) = FALSE
   THEN
       #i := 0;

       WHILE #i < "pq_size"(#self) DO
           IF "gi_compare_vehicle_numbers"(vehicle_number_1 := #vehicle_number, vehicle_number_2 := #self.queue_array[#i].glass.vehicle_number) = TRUE
           THEN
               #pq_find_by_vehicle_number := #i;
               RETURN;
           END_IF;

           #i := #i + 1;
       END_WHILE;
   END_IF;
END_FUNCTION

FUNCTION "pq_clear" : Void   // FC25, SCL
{ S7_Optimized_Access := 'TRUE' }
VERSION : 0.1
// Initialize all assigned items of array to default value, but for optimization purpose, all data inside glass_info struct are not deleted until next write operation when will be rewrited
   VAR_IN_OUT
      self : "PriorityQueue";
   END_VAR
   VAR_TEMP
      i : Int;
   END_VAR
BEGIN

   WHILE #i < "pq_size"(#self) DO
       #self.queue_array[#i].allocated := false;
       #self.queue_array[#i].priority := false;

       #i := #i + 1;
   END_WHILE;

   #self.size := 0;
END_FUNCTION

FUNCTION "pg_shift_right" : Void   // FC30, SCL
{ S7_Optimized_Access := 'TRUE' }
VERSION : 0.1
// Shifts all records in array one position to right
   VAR_IN_OUT
      self : "PriorityQueue";
   END_VAR
   VAR_TEMP
      i : Int;
   END_VAR
BEGIN

   IF "pq_size"(#self) >= 2
   THEN
       #i := "pq_size"(#self);

       WHILE #i > 0 DO
           #self.queue_array[#i] := #self.queue_array[#i - 1];
           #i := #i - 1;
       END_WHILE;
   END_IF;
END_FUNCTION

FUNCTION "pg_shift_left" : Void   // FC31, SCL
{ S7_Optimized_Access := 'TRUE' }
VERSION : 0.1
// Shifts all records in array one position to left
   VAR_IN_OUT
      self : "PriorityQueue";
   END_VAR
   VAR_TEMP
      i : Int;
   END_VAR
BEGIN
   #i := 0;

   IF "pq_size"(#self) >= 2
   THEN
       WHILE #i < "pq_size"(#self) - 1 DO
           #self.queue_array[#i] := #self.queue_array[#i + 1];
           #i := #i + 1;
       END_WHILE;
   END_IF;
END_FUNCTION

// folder: Valve/Valve2Pos

FUNCTION "valve_2_pos_control" : Void   // FC49, SCL
{ S7_Optimized_Access := 'TRUE' }
VERSION : 0.1
   VAR_INPUT
      reaction_delay : Time;
   END_VAR
   VAR_IN_OUT
      self : "Valve2Pos";
      io : "IOValve2pos";
   END_VAR
BEGIN

   #self.reaction_delay := #reaction_delay;

   "valve_2_pos_watchdog_timer"(#self);
   "valve_2_pos_synchronize_internal_request_signals"(#self);

   (*
   ** synchronization of output signals with internal logic states
   *)
   #io.o_end_position := #self.cmd_end_position AND #self.request_release = false;
   #io.o_start_position := #self.cmd_start_position AND #self.request_release = false;
END_FUNCTION

// folder: Valve/Valve2Pos/api

FUNCTION "valve_2_pos_set_end_position" : Void   // FC59, SCL
{ S7_Optimized_Access := 'TRUE' }
VERSION : 0.1
   VAR_IN_OUT
      self : "Valve2Pos";
   END_VAR
BEGIN


   #self.cmd_end_position := true;
   #self.cmd_start_position := false;
END_FUNCTION

FUNCTION "valve_2_pos_set_start_position" : Void   // FC60, SCL
{ S7_Optimized_Access := 'TRUE' }
VERSION : 0.1
   VAR_IN_OUT
      self : "Valve2Pos";
   END_VAR
BEGIN


   #self.cmd_end_position := false;
   #self.cmd_start_position := true;
END_FUNCTION

FUNCTION "valve_2_pos_is_end_position" : Bool   // FC69, SCL
{ S7_Optimized_Access := 'TRUE' }
VERSION : 0.1
   VAR_IN_OUT
      self : "Valve2Pos";
   END_VAR
BEGIN


   #valve_2_pos_is_end_position := #self.io.i_end_position;
END_FUNCTION

FUNCTION "valve_2_pos_is_start_position" : Bool   // FC70, SCL
{ S7_Optimized_Access := 'TRUE' }
VERSION : 0.1
   VAR_IN_OUT
      self : "Valve2Pos";
   END_VAR
BEGIN


   #valve_2_pos_is_start_position := #self.io.i_start_position;
END_FUNCTION

FUNCTION "valve_2_pos_set_release" : Void   // FC72, SCL
{ S7_Optimized_Access := 'TRUE' }
VERSION : 0.1
   VAR_INPUT
      release : Bool;
   END_VAR
   VAR_IN_OUT
      self : "Valve2Pos";
   END_VAR
BEGIN


   #self.request_release := #release;
END_FUNCTION

// folder: Valve/Valve2Pos/fce

FUNCTION "valve_2_pos_set_internal_logic_signal" : Void   // FC50, SCL
{ S7_Optimized_Access := 'TRUE' }
VERSION : 0.1
   VAR_INPUT
      request_A : Bool;
      request_B : Bool;
   END_VAR
   VAR_IN_OUT
      signal_A : Bool;
      signal_B : Bool;
   END_VAR
BEGIN

   IF #request_A = true
       AND #request_B = FALSE
   THEN
       #signal_A := true;
       #signal_B := false;
   END_IF;
END_FUNCTION

FUNCTION "valve_2_pos_watchdog_timer" : Void   // FC51, SCL
{ S7_Optimized_Access := 'TRUE' }
VERSION : 0.1
   VAR_IN_OUT
      self : "Valve2Pos";
   END_VAR
   VAR_TEMP
      watchdog_enable : Bool;
      error_start_position : Bool;
      error_end_position : Bool;
      error_position_sensors : Bool;
   END_VAR
BEGIN

   #error_end_position := (#self.cmd_end_position = true AND #self.io.i_end_position = false);
   #error_start_position := (#self.cmd_start_position = true AND #self.io.i_start_position = false);
   #error_position_sensors := (#self.io.i_end_position = true AND #self.io.i_start_position = true);

   #watchdog_enable := #self.request_release = false AND (#error_end_position OR #error_position_sensors OR #error_start_position);

   #self.watchdog_timer(PT := #self.reaction_delay, IN := #watchdog_enable);

   IF #watchdog_enable = false
   THEN
       RESET_TIMER(#self.watchdog_timer);
   END_IF;

   #self.status_error := #self.watchdog_timer.Q;
END_FUNCTION

FUNCTION "valve_2_pos_synchronize_internal_request_signals" : Void   // FC52, SCL
{ S7_Optimized_Access := 'TRUE' }
VERSION : 0.1
   VAR_IN_OUT
      self : "Valve2Pos";
   END_VAR
BEGIN


   "valve_2_pos_set_internal_logic_signal"(request_A := #self.request_signal_end,
                                     request_B := #self.request_signal_start,
                                     signal_A := #self.cmd_end_position,
                                     signal_B := #self.cmd_start_position);

   "valve_2_pos_set_internal_logic_signal"(request_A := #self.request_signal_start,
                                     request_B := #self.request_signal_end,
                                     signal_A := #self.cmd_start_position,
                                     signal_B := #self.cmd_end_position);

   IF #self.request_release = TRUE
   THEN
       #self.cmd_end_position := false;
       #self.cmd_start_position := false;
   END_IF;
END_FUNCTION

// folder: io

FUNCTION_BLOCK "io_sync"   // FB2, SCL
{ S7_Optimized_Access := 'TRUE' }
VERSION : 0.1
   VAR
      test_valve_io : "IOValve2pos";
      test_curing_buffer_io : "IOCuringBuffer";
      test_centering_bed_io : "IOCenterngBed";
   END_VAR
BEGIN

   #test_valve_io.i_end_position := "i_test_vavlve_end";
   #test_valve_io.i_start_position := "i_test_valve_start";


   "o_test_valve_end" := #test_valve_io.o_end_position;
   "o_test_valve_start" := #test_valve_io.o_start_position;
END_FUNCTION_BLOCK

// folder: unitLib

FUNCTION_BLOCK "PLCUnitLib"   // FB1, SCL
{ S7_Optimized_Access := 'TRUE' }
VERSION : 0.1
   VAR
      TCON_Instance : TCON;
      TDISCON_Instance : TDISCON;
      TRCV_Instance : TRCV;
      TSEND_Instance : TSEND;
      self : "UnitLib";
   END_VAR
   VAR CONSTANT
      id : Conn_Ouc := 1;
   END_VAR
BEGIN

   "network"("TCON_":=#TCON_Instance,
             "TDISCON_":=#TDISCON_Instance,
             "TRCV_":=#TRCV_Instance,
             "TSEND_":=#TSEND_Instance,
             self:= #self);

   IF #self.step = 0
   THEN
       IF #TCON_Instance.DONE = true
       THEN
           #self.step := 1;
       END_IF;
   ELSIF #self.step = 1
   THEN
       IF #TRCV_Instance.NDR = true
       THEN
           #self.step := 2;
       END_IF;
   ELSIF #self.step = 2
   THEN
       "communication"(#self);
       #self.step := 3;

   ELSIF #self.step = 3
   THEN
       IF #TSEND_Instance.DONE = true
       THEN
           #self.step := 1;
       END_IF;
   ELSE
       IF #TDISCON_Instance.DONE = true
           OR #TDISCON_Instance.ERROR = true
       THEN
           #self.step := 0;
       END_IF;
   END_IF;


   IF #TSEND_Instance.ERROR = true
   THEN
       #self.step := 4;
   END_IF;
END_FUNCTION_BLOCK

FUNCTION "test_runtime" : Bool   // FC1, SCL
{ S7_Optimized_Access := 'TRUE' }
VERSION : 0.1
   VAR_INPUT
      ts_index : Byte;
      tc_index : Byte;
   END_VAR
   VAR_IN_OUT
      self : "UnitLib";
   END_VAR
BEGIN



   IF #ts_index = 1
   THEN
       (* priority queue tests *)
       IF #tc_index = 1
       THEN
           #test_runtime := "pq_enqueue_test"();
       ELSIF #tc_index = 2
       THEN
           #test_runtime := "pq_size_test"();
       ELSIF #tc_index = 3
       THEN
           #test_runtime := "pq_is_empty_test"();
       ELSIF #tc_index = 4
       THEN
           #test_runtime := "pq_peek_test"();
       ELSIF #tc_index = 5
       THEN
           #test_runtime := "pq_delete_by_index_test"();
       ELSIF #tc_index = 6
       THEN
           #test_runtime := "pq_dequeue_test"();
       ELSIF #tc_index = 7
       THEN
           #test_runtime := "pq_find_by_vehicle_number_test"();
       ELSIF #tc_index = 8
       THEN
           #test_runtime := "pq_clear_test"();
       ELSE
           #test_runtime := false;
       END_IF;
   ELSIF #ts_index = 2
   THEN
       (* curring buffer tests *)
       IF #tc_index = 1
       THEN
           #test_runtime := "cb_get_class_info_test"();
       ELSIF #tc_index = 2
       THEN
           #test_runtime := "cb_insert_glass_test"();
       ELSIF #tc_index = 3
       THEN
           #test_runtime := "cb_is_drawer_enabled_test"();
       ELSIF #tc_index = 4
       THEN
           #test_runtime := "cb_is_drawer_free_test"();
       ELSIF #tc_index = 5
       THEN
           #test_runtime := "cb_is_glass_expired_test"();
       ELSIF #tc_index = 6
       THEN
           #test_runtime := "cb_is_glass_ready_test"();
       ELSIF #tc_index = 7
       THEN
           #test_runtime := "cb_remove_glass_test"();
       ELSE
           #test_runtime := false;
       END_IF;
   ELSIF #ts_index = 3
   THEN
       IF #tc_index = 1
       THEN
           #test_runtime := "centering_bed_do_centering_test"();
       ELSIF #tc_index = 2
       THEN
           #test_runtime := "centering_bed_get_state_test"();
       ELSIF #tc_index = 3
       THEN
           #test_runtime := "centering_bed_is_centered_test"();
       ELSIF #tc_index = 4
       THEN
           #test_runtime := "centering_bed_is_occupied_test"();
       ELSIF #tc_index = 5
       THEN
           #test_runtime := "centering_bed_release_centering_test"();
       ELSE
           #test_runtime := false;
       END_IF;
   ELSE
       #test_runtime := false;
   END_IF;
END_FUNCTION

FUNCTION "network" : Void   // FC2, SCL
{ S7_Optimized_Access := 'TRUE' }
VERSION : 0.1
   VAR_IN_OUT
      TCON_ : TCON;
      TDISCON_ : TDISCON;
      TRCV_ : TRCV;
      TSEND_ : TSEND;
      self : "UnitLib";
   END_VAR
BEGIN



   #"TCON_"(CONNECT := "PLC_1_Connection_DB",
            REQ := #self.step = 0,
            ID := #self.network_id);

   #"TRCV_"(ID := #self.network_id,
                  EN_R := true,
                  LEN := 0,
                  ADHOC := true,
                  DATA := #self.#input_buffer);

   #"TSEND_"(ID := #self.network_id,
                   LEN := #self.output_len,
                   REQ := #self.step = 3,
                   DATA := #self.output_buffer);

   #"TDISCON_"(REQ := (NOT #"TDISCON_".REQ) AND (#self.step > 3),
               ID := #self.network_id);
END_FUNCTION

FUNCTION "communication" : Void   // FC10, SCL
{ S7_Optimized_Access := 'TRUE' }
VERSION : 0.1
   VAR_IN_OUT
      self : "UnitLib";
   END_VAR
BEGIN
   IF #self.input_buffer[0] = 1
   THEN
       "unit_lib_build_ping_response"(#self);
   ELSIF #self.input_buffer[0] = 2
   THEN
       "unit_lib_build_reset_response"(#self);
   ELSIF #self.input_buffer[0] = 3
   THEN
       "unit_lib_build_ts_count_response"(#self);
   ELSIF #self.input_buffer[0] = 4
   THEN
       "unit_lib_build_tc_count_response"(#self);
   ELSIF #self.input_buffer[0] = 5
   THEN
       "unit_lib_build_ts_name_response"(#self);
   ELSIF #self.input_buffer[0] = 6
   THEN
       "unit_lib_build_tc_name_response"(#self);
   ELSIF #self.input_buffer[0] = 7
   THEN
       "unit_lib_build_run_test_response"(#self);
   ELSE
       #self.output_len := 1;
       #self.output_buffer[0] := 255;
   END_IF;
END_FUNCTION

// folder: unitLib/cmd

FUNCTION "unit_lib_build_ping_response" : Void   // FC3, SCL
{ S7_Optimized_Access := 'TRUE' }
VERSION : 0.1
   VAR_IN_OUT
      self : "UnitLib";
   END_VAR
BEGIN
   #self.output_buffer[0] := 1;
   #self.output_buffer[1] := 1;
   #self.output_len := 2;
END_FUNCTION

FUNCTION "unit_lib_build_reset_response" : Void   // FC4, SCL
{ S7_Optimized_Access := 'TRUE' }
VERSION : 0.1
   VAR_IN_OUT
      self : "UnitLib";
   END_VAR
BEGIN
   #self.output_len := 2;
   #self.output_buffer[0] := 2;
   #self.output_buffer[1] := 1;
END_FUNCTION

FUNCTION "unit_lib_build_ts_count_response" : Void   // FC5, SCL
{ S7_Optimized_Access := 'TRUE' }
VERSION : 0.1
   VAR_IN_OUT
      self : "UnitLib";
   END_VAR
BEGIN
   #self.output_len := 2;
   #self.output_buffer[0] := 3;
   #self.output_buffer[1] := #self.ts_size;
END_FUNCTION

FUNCTION "unit_lib_build_tc_count_response" : Void   // FC6, SCL
{ S7_Optimized_Access := 'TRUE' }
VERSION : 0.1
   VAR_IN_OUT
      self : "UnitLib";
   END_VAR
BEGIN
   #self.output_len := 2;
   #self.output_buffer[0] := 4;
   #self.output_buffer[1] := #self.unit[#self.input_buffer[1]].tc_size;
END_FUNCTION

FUNCTION "unit_lib_build_ts_name_response" : Void   // FC7, SCL
{ S7_Optimized_Access := 'TRUE' }
VERSION : 0.1
   VAR_IN_OUT
      self : "UnitLib";
   END_VAR
   VAR_TEMP
      i : Int;
      name_array : Array[1..128] of Char;
      cnt : Int;
   END_VAR
BEGIN

   #self.output_buffer[0] := 5;

   #i := 1;
   #cnt := LEN(#self.unit[#self.input_buffer[1]].ts_name) + 1;

   WHILE #i < LEN(#self.unit[#self.input_buffer[1]].ts_name) + 1
   DO
       #self.output_buffer[#i] := #self.unit[#self.input_buffer[1]].ts_name[#i];
       #i := #i + 1;
   END_WHILE;

   #self.output_buffer[#i] := 0;

   #self.output_len := INT_TO_BYTE(#cnt);
END_FUNCTION

FUNCTION "unit_lib_build_tc_name_response" : Void   // FC8, SCL
{ S7_Optimized_Access := 'TRUE' }
VERSION : 0.1
   VAR_IN_OUT
      self : "UnitLib";
   END_VAR
   VAR_TEMP
      i : Int;
      name_array : Array[1..128] of Char;
      cnt : Int;
      "name" : String;
   END_VAR
BEGIN
   #self.output_len := 2;
   #self.output_buffer[0] := 6;


   #i := 1;
   #name := #self.unit[#self.input_buffer[1]].tc_name[#self.input_buffer[2]];
   #cnt := LEN(#name) + 1;

   WHILE #i < #cnt
   DO
       #self.output_buffer[#i] := #name[#i];
       #i := #i + 1;
   END_WHILE;

   #self.output_buffer[#i] := 0;
   #self.output_len := INT_TO_BYTE(#cnt);
END_FUNCTION

FUNCTION "unit_lib_build_run_test_response" : Void   // FC9, SCL
{ S7_Optimized_Access := 'TRUE' }
VERSION : 0.1
   VAR_IN_OUT
      self : "UnitLib";
   END_VAR
BEGIN
   #self.output_len := 2;
   #self.output_buffer[0] := 7;



   IF "test_runtime"(ts_index:=#self.input_buffer[1], tc_index:=#self.input_buffer[2], self:=#self) = true THEN
       #self.output_buffer[1] := 1;
   ELSE
       #self.output_buffer[1] := 0;
   END_IF;
END_FUNCTION

// folder: unitLib/test_suites/centering_bed_test

FUNCTION "centering_bed_is_centered_test" : Bool   // FC61, SCL
{ S7_Optimized_Access := 'TRUE' }
VERSION : 0.1
BEGIN


   #centering_bed_is_centered_test := false;
END_FUNCTION

FUNCTION "centering_bed_do_centering_test" : Bool   // FC62, SCL
{ S7_Optimized_Access := 'TRUE' }
VERSION : 0.1
BEGIN


   #centering_bed_do_centering_test := false;
END_FUNCTION

FUNCTION "centering_bed_is_occupied_test" : Bool   // FC63, SCL
{ S7_Optimized_Access := 'TRUE' }
VERSION : 0.1
BEGIN


   #centering_bed_is_occupied_test := false;
END_FUNCTION

FUNCTION "centering_bed_get_state_test" : Bool   // FC64, SCL
{ S7_Optimized_Access := 'TRUE' }
VERSION : 0.1
BEGIN



   #centering_bed_get_state_test := false;
END_FUNCTION

FUNCTION "centering_bed_release_centering_test" : Bool   // FC65, SCL
{ S7_Optimized_Access := 'TRUE' }
VERSION : 0.1
BEGIN


   #centering_bed_release_centering_test := false;
END_FUNCTION

// folder: unitLib/test_suites/curing_buffer_test

FUNCTION "cb_insert_glass_test" : Bool   // FC38, SCL
{ S7_Optimized_Access := 'TRUE' }
VERSION : 0.1
   VAR_TEMP
      glass1 : "GlassInfo";
      glass2 : "GlassInfo";
      empty_glass : "GlassInfo";
      time_ : DTL;
   END_VAR
BEGIN


   "DB_process_data".curing_buffer_1.drawer_array[0].enable := true;
   #glass1 := "gi_new"(rear_window := 'VW-Number', vehicle_model := 'T7', vehicle_number := '123456789 00');
   #glass2 := "gi_new"(rear_window := 'VW-Number', vehicle_model := 'T7', vehicle_number := '123456790 00');

   IF "cb_insert_glass"(drawer_index := 0, glass := #glass1, self := "DB_process_data".curing_buffer_1) = TRUE
       AND "cb_insert_glass"(drawer_index := 0, glass := #glass2, self := "DB_process_data".curing_buffer_1) = FALSE
   THEN
       IF "DB_process_data".curing_buffer_1.drawer_array[0].occupied
           AND "DB_process_data".curing_buffer_1.drawer_array[0].glass.rear_window = 'VW-Number'
           AND "DB_process_data".curing_buffer_1.drawer_array[0].glass.vehicle_model = 'T7'
           AND "DB_process_data".curing_buffer_1.drawer_array[0].glass.vehicle_number = '123456789 00'
           AND "DB_process_data".curing_buffer_1.drawer_array[0].insertion_time <> #"time_"
       THEN
           #cb_insert_glass_test := true;
       ELSE
           #cb_insert_glass_test := false;
       END_IF;
   ELSE
       #cb_insert_glass_test := false;
   END_IF;

   "DB_process_data".curing_buffer_1.drawer_array[0].enable := false;
   "DB_process_data".curing_buffer_1.drawer_array[0].glass := #empty_glass;
   "DB_process_data".curing_buffer_1.drawer_array[0].occupied := false;
   "DB_process_data".curing_buffer_1.drawer_array[0].insertion_time := #"time_";
   "clear_curing_buffer"();
END_FUNCTION

FUNCTION "cb_is_drawer_free_test" : Bool   // FC39, SCL
{ S7_Optimized_Access := 'TRUE' }
VERSION : 0.1
BEGIN

   "insert_some_glass"();
   "DB_process_data".curing_buffer_1.drawer_array[3].enable := true;
   "DB_process_data".curing_buffer_1.drawer_array[2].enable := true;
   "DB_process_data".curing_buffer_1.drawer_array[2].presence_sensor := true;

   IF "cb_is_drawer_free"(drawer_index := 0, self := "DB_process_data".curing_buffer_1) = FALSE
       AND "cb_is_drawer_free"(drawer_index := 1, self := "DB_process_data".curing_buffer_1) = FALSE
       AND "cb_is_drawer_free"(drawer_index := 2, self := "DB_process_data".curing_buffer_1) = FALSE
       AND "cb_is_drawer_free"(drawer_index := 3, self := "DB_process_data".curing_buffer_1) = true
   THEN
       #cb_is_drawer_free_test := true;
   ELSE
       #cb_is_drawer_free_test := false;
   END_IF;

   "DB_process_data".curing_buffer_1.drawer_array[3].enable := false;
   "DB_process_data".curing_buffer_1.drawer_array[2].enable := false;
   "DB_process_data".curing_buffer_1.drawer_array[2].presence_sensor := false;

   "clear_curing_buffer"();
END_FUNCTION

FUNCTION "cb_is_drawer_enabled_test" : Bool   // FC40, SCL
{ S7_Optimized_Access := 'TRUE' }
VERSION : 0.1
BEGIN

   "DB_process_data".curing_buffer_1.drawer_array[0].enable := true;

   IF "cb_is_drawer_enabled"(drawer_index := 0, self := "DB_process_data".curing_buffer_1) = TRUE
       AND "cb_is_drawer_enabled"(drawer_index := 1, self := "DB_process_data".curing_buffer_1) = FALSE
   THEN
       #cb_is_drawer_enabled_test := true;
   ELSE
       #cb_is_drawer_enabled_test := false;
   END_IF;

   "DB_process_data".curing_buffer_1.drawer_array[0].enable := false;
END_FUNCTION

FUNCTION "cb_remove_glass_test" : Bool   // FC41, SCL
{ S7_Optimized_Access := 'TRUE' }
VERSION : 0.1
BEGIN
   "insert_some_glass"();

   IF "cb_is_drawer_free"(drawer_index := 0, self := "DB_process_data".curing_buffer_1) = FALSE
   THEN
       IF "cb_remove_glass"(drawer_index := 0, self := "DB_process_data".curing_buffer_1) = TRUE
       THEN
           IF "cb_is_drawer_free"(drawer_index := 0, self := "DB_process_data".curing_buffer_1) = TRUE
           THEN
               #cb_remove_glass_test := true;
           ELSE
               #cb_remove_glass_test := false;
           END_IF;
       ELSE
           #cb_remove_glass_test := false;
       END_IF;
   ELSE

       #cb_remove_glass_test := false;
   END_IF;


   "clear_curing_buffer"();
END_FUNCTION

FUNCTION "cb_is_glass_expired_test" : Bool   // FC42, SCL
{ S7_Optimized_Access := 'TRUE' }
VERSION : 0.1
   VAR_TEMP
      test_current_time : DTL;
      return_val : Int;
   END_VAR
   VAR CONSTANT
      min_expiration_time : Time := T#10m;
      max_expiration_time : Time := T#8h;
      min_expiration_time_empty : Time;
      max_expiration_time_empty : Time;
      test_ready_time : Time := T#4h;
      test_expiration_time : Time := T#10h;
      test_not_ready_time : Time := T#5m;
      empty_time : DTL;
   END_VAR
BEGIN

   "DB_process_data".curing_buffer_1.max_expiration_time := #max_expiration_time;
   "DB_process_data".curing_buffer_1.min_expiration_time := #min_expiration_time;

   #return_val := RD_SYS_T(#test_current_time);

   "DB_process_data".curing_buffer_1.drawer_array[0].enable := true;
   "DB_process_data".curing_buffer_1.drawer_array[1].enable := true;
   "DB_process_data".curing_buffer_1.drawer_array[2].enable := true;

   "DB_process_data".curing_buffer_1.drawer_array[0].occupied := true;
   "DB_process_data".curing_buffer_1.drawer_array[1].occupied := true;
   "DB_process_data".curing_buffer_1.drawer_array[2].occupied := true;


   "DB_process_data".curing_buffer_1.drawer_array[0].insertion_time := T_SUB(IN1:=#test_current_time, IN2:=#test_ready_time);
   "DB_process_data".curing_buffer_1.drawer_array[1].insertion_time := T_SUB(IN1 := #test_current_time, IN2 := #test_expiration_time);
   "DB_process_data".curing_buffer_1.drawer_array[2].insertion_time := T_SUB(IN1 := #test_current_time, IN2 := #test_not_ready_time);
   "DB_process_data".curing_buffer_1.drawer_array[3].insertion_time := T_SUB(IN1 := #test_current_time, IN2 := #test_ready_time);

   IF "cb_is_glass_expired"(drawer_index := 0, self := "DB_process_data".curing_buffer_1) = TRUE
       AND "cb_is_glass_expired"(drawer_index := 1, self := "DB_process_data".curing_buffer_1) = FALSE
       AND "cb_is_glass_expired"(drawer_index := 2, self := "DB_process_data".curing_buffer_1) = true
       AND "cb_is_glass_expired"(drawer_index := 3, self := "DB_process_data".curing_buffer_1) = false
   THEN
       #cb_is_glass_expired_test := true;
   ELSE

       #cb_is_glass_expired_test := false;
   END_IF;


   "DB_process_data".curing_buffer_1.drawer_array[0].enable := false;
   "DB_process_data".curing_buffer_1.drawer_array[1].enable := false;
   "DB_process_data".curing_buffer_1.drawer_array[2].enable := false;

   "DB_process_data".curing_buffer_1.drawer_array[0].occupied := false;
   "DB_process_data".curing_buffer_1.drawer_array[1].occupied := false;
   "DB_process_data".curing_buffer_1.drawer_array[2].occupied := false;

   "DB_process_data".curing_buffer_1.drawer_array[0].insertion_time := #empty_time;
   "DB_process_data".curing_buffer_1.drawer_array[1].insertion_time := #empty_time;
   "DB_process_data".curing_buffer_1.drawer_array[2].insertion_time := #empty_time;
   "DB_process_data".curing_buffer_1.drawer_array[3].insertion_time := #empty_time;

   "DB_process_data".curing_buffer_1.max_expiration_time := #max_expiration_time_empty;
   "DB_process_data".curing_buffer_1.min_expiration_time := #min_expiration_time_empty;
END_FUNCTION

FUNCTION "cb_get_class_info_test" : Bool   // FC43, SCL
{ S7_Optimized_Access := 'TRUE' }
VERSION : 0.1
   VAR_TEMP
      glass : "GlassInfo";
   END_VAR
BEGIN
   "insert_some_glass"();

   IF "cb_is_drawer_enabled"(drawer_index := 0, self := "DB_process_data".curing_buffer_1) = true
       AND "cb_is_drawer_free"(drawer_index := 0, self := "DB_process_data".curing_buffer_1) = false
   THEN
       #glass := "cb_get_class_info"(drawer_index := 0, self := "DB_process_data".curing_buffer_1);

       IF #glass.vehicle_number = '123456789 00'
           AND #glass.rear_window = 'VW-Number'
           AND #glass.vehicle_model = 'T7'
       THEN
           #cb_get_class_info_test := true;
       ELSE
           #cb_get_class_info_test := false;
       END_IF;
   ELSE
       #cb_get_class_info_test := false;
   END_IF;

   "clear_curing_buffer"();
END_FUNCTION

FUNCTION "cb_is_glass_ready_test" : Bool   // FC48, SCL
{ S7_Optimized_Access := 'TRUE' }
VERSION : 0.1
   VAR_TEMP
      test_current_time : DTL;
      return_val : Int;
   END_VAR
   VAR CONSTANT
      min_expiration_time : Time := T#10m;
      max_expiration_time : Time := T#8h;
      min_expiration_time_empty : Time;
      max_expiration_time_empty : Time;
      test_ready_time : Time := T#4h;
      test_expiration_time : Time := T#10h;
      test_not_ready_time : Time := T#5m;
      empty_time : DTL;
   END_VAR
BEGIN



   "DB_process_data".curing_buffer_1.max_expiration_time := #max_expiration_time;
   "DB_process_data".curing_buffer_1.min_expiration_time := #min_expiration_time;

   #return_val := RD_SYS_T(#test_current_time);

   "DB_process_data".curing_buffer_1.drawer_array[0].enable := true;
   "DB_process_data".curing_buffer_1.drawer_array[1].enable := true;
   "DB_process_data".curing_buffer_1.drawer_array[2].enable := true;

   "DB_process_data".curing_buffer_1.drawer_array[0].occupied := true;
   "DB_process_data".curing_buffer_1.drawer_array[1].occupied := true;
   "DB_process_data".curing_buffer_1.drawer_array[2].occupied := true;


   "DB_process_data".curing_buffer_1.drawer_array[0].insertion_time := T_SUB(IN1 := #test_current_time, IN2 := #test_ready_time);
   "DB_process_data".curing_buffer_1.drawer_array[1].insertion_time := T_SUB(IN1 := #test_current_time, IN2 := #test_expiration_time);
   "DB_process_data".curing_buffer_1.drawer_array[2].insertion_time := T_SUB(IN1 := #test_current_time, IN2 := #test_not_ready_time);
   "DB_process_data".curing_buffer_1.drawer_array[3].insertion_time := T_SUB(IN1 := #test_current_time, IN2 := #test_ready_time);

   IF "cb_is_glass_ready"(drawer_index := 0, self := "DB_process_data".curing_buffer_1) = TRUE
       AND "cb_is_glass_ready"(drawer_index := 1, self := "DB_process_data".curing_buffer_1) = true
       AND "cb_is_glass_ready"(drawer_index := 2, self := "DB_process_data".curing_buffer_1) = false
       AND "cb_is_glass_ready"(drawer_index := 3, self := "DB_process_data".curing_buffer_1) = false
   THEN
       #cb_is_glass_ready_test := true;
   ELSE

       #cb_is_glass_ready_test := false;
   END_IF;


   "DB_process_data".curing_buffer_1.drawer_array[0].enable := false;
   "DB_process_data".curing_buffer_1.drawer_array[1].enable := false;
   "DB_process_data".curing_buffer_1.drawer_array[2].enable := false;

   "DB_process_data".curing_buffer_1.drawer_array[0].occupied := false;
   "DB_process_data".curing_buffer_1.drawer_array[1].occupied := false;
   "DB_process_data".curing_buffer_1.drawer_array[2].occupied := false;

   "DB_process_data".curing_buffer_1.drawer_array[0].insertion_time := #empty_time;
   "DB_process_data".curing_buffer_1.drawer_array[1].insertion_time := #empty_time;
   "DB_process_data".curing_buffer_1.drawer_array[2].insertion_time := #empty_time;
   "DB_process_data".curing_buffer_1.drawer_array[3].insertion_time := #empty_time;

   "DB_process_data".curing_buffer_1.max_expiration_time := #max_expiration_time_empty;
   "DB_process_data".curing_buffer_1.min_expiration_time := #min_expiration_time_empty;
END_FUNCTION

// folder: unitLib/test_suites/curing_buffer_test/cb_test_util

FUNCTION "insert_some_glass" : Void   // FC45, SCL
{ S7_Optimized_Access := 'TRUE' }
VERSION : 0.1
   VAR_TEMP
      glass1 : "GlassInfo";
      glass2 : "GlassInfo";
      glass3 : "GlassInfo";
      return_ : Bool;
   END_VAR
BEGIN

   "DB_process_data".curing_buffer_1.drawer_array[0].enable := true;
   "DB_process_data".curing_buffer_1.drawer_array[1].enable := true;
   "DB_process_data".curing_buffer_1.drawer_array[2].enable := true;

   #glass1 := "gi_new"(rear_window := 'VW-Number', vehicle_model := 'T7', vehicle_number := '123456789 00');
   #glass2 := "gi_new"(rear_window := 'VW-Number', vehicle_model := 'T7', vehicle_number := '123456790 00');
   #glass3 := "gi_new"(rear_window := 'VW-Number', vehicle_model := 'T7', vehicle_number := '123456791 00');

   #"return_" := "cb_insert_glass"(drawer_index := 0, glass := #glass1, self := "DB_process_data".curing_buffer_1);
   #"return_" := "cb_insert_glass"(drawer_index := 1, glass := #glass2, self := "DB_process_data".curing_buffer_1);
   #"return_" := "cb_insert_glass"(drawer_index := 2, glass := #glass2, self := "DB_process_data".curing_buffer_1);
END_FUNCTION

FUNCTION "clear_curing_buffer" : Void   // FC46, SCL
{ S7_Optimized_Access := 'TRUE' }
VERSION : 0.1
   VAR_TEMP
      glass : "GlassInfo";
      time_ : DTL;
   END_VAR
BEGIN
   "DB_process_data".curing_buffer_1.drawer_array[0].enable := false;
   "DB_process_data".curing_buffer_1.drawer_array[1].enable := false;
   "DB_process_data".curing_buffer_1.drawer_array[2].enable := false;

   "DB_process_data".curing_buffer_1.drawer_array[0].glass := #glass;
   "DB_process_data".curing_buffer_1.drawer_array[1].glass := #glass;
   "DB_process_data".curing_buffer_1.drawer_array[2].glass := #glass;

   "DB_process_data".curing_buffer_1.drawer_array[0].occupied := false;
   "DB_process_data".curing_buffer_1.drawer_array[1].occupied := false;
   "DB_process_data".curing_buffer_1.drawer_array[2].occupied := false;


   "DB_process_data".curing_buffer_1.drawer_array[0].insertion_time := #"time_";
   "DB_process_data".curing_buffer_1.drawer_array[1].insertion_time := #"time_";
   "DB_process_data".curing_buffer_1.drawer_array[2].insertion_time := #"time_";
END_FUNCTION

// folder: unitLib/test_suites/priority_queue_test

FUNCTION "pq_clear_test" : Bool   // FC17, SCL
{ S7_Optimized_Access := 'TRUE' }
VERSION : 0.1
BEGIN


   "fill_priority_queue"();


   IF "pq_size"("DB_process_data".glass_queue) > 0
   THEN
       "pq_clear"("DB_process_data".glass_queue);

       IF "pq_is_empty"("DB_process_data".glass_queue) = TRUE
           AND "pq_size"("DB_process_data".glass_queue) = 0
       THEN
           #pq_clear_test := true;
       ELSE
           #pq_clear_test := false;
       END_IF;
   ELSE
       #pq_clear_test := false;
   END_IF;
END_FUNCTION

FUNCTION "pq_enqueue_test" : Bool   // FC19, SCL
{ S7_Optimized_Access := 'TRUE' }
VERSION : 0.1
   VAR_TEMP
      size_before : Int;
      size_after : Int;
      glass_ordinary1 : "GlassInfo";
      glass_ordinary2 : "GlassInfo";
      glass_priority : "GlassInfo";
      glass_duplicit : "GlassInfo";
      ret_val_1 : Bool;
   END_VAR
BEGIN

   IF "pq_is_empty"("DB_process_data".glass_queue) = TRUE
   THEN
       #size_before := "pq_size"("DB_process_data".glass_queue);

       #glass_ordinary1 := "gi_new"(rear_window := 'VW-0001', vehicle_model := 'IDBuzz', vehicle_number := '123456789 00');
       #glass_ordinary2 := "gi_new"(rear_window := 'VW-0001', vehicle_model := 'IDBuzz', vehicle_number := '123456790 00');
       #glass_priority := "gi_new"(rear_window := 'VW-0001', vehicle_model := 'T7', vehicle_number := '123456791 00');
       #glass_duplicit := "gi_new"(rear_window := 'VW-0001', vehicle_model := 'IDBuzz', vehicle_number := '123456790 01');

       IF "pq_enqueue"(glass:=#glass_ordinary1, priority:=false, self:="DB_process_data".glass_queue) = true
           AND "pq_enqueue"(glass := #glass_ordinary2, priority := false, self := "DB_process_data".glass_queue) = true
           AND "pq_enqueue"(glass := #glass_priority, priority := true, self := "DB_process_data".glass_queue) = true
           AND "pq_enqueue"(glass := #glass_duplicit, priority := false, self := "DB_process_data".glass_queue) = true
       THEN
           #size_after := "pq_size"("DB_process_data".glass_queue);

           IF #size_before = #size_after - 3
               AND "DB_process_data".glass_queue.queue_array[0].allocated = true
               AND "DB_process_data".glass_queue.queue_array[1].allocated = true
               AND "DB_process_data".glass_queue.queue_array[2].allocated = true
               AND "DB_process_data".glass_queue.queue_array[0].priority = TRUE
               AND "DB_process_data".glass_queue.queue_array[1].priority = false
               AND "DB_process_data".glass_queue.queue_array[2].priority = FALSE
               AND "DB_process_data".glass_queue.queue_array[0].glass.vehicle_number = '123456791 00'
               AND "DB_process_data".glass_queue.queue_array[1].glass.vehicle_number = '123456789 00'
               AND "DB_process_data".glass_queue.queue_array[2].glass.vehicle_number = '123456790 01'
           THEN
               #pq_enqueue_test := true;
           ELSE
               #pq_enqueue_test := false;
           END_IF;

           "pq_clear"("DB_process_data".glass_queue);
       ELSE
           #pq_enqueue_test := false;
       END_IF;
   ELSE
       #pq_enqueue_test := false;
   END_IF;
END_FUNCTION

FUNCTION "pq_dequeue_test" : Bool   // FC20, SCL
{ S7_Optimized_Access := 'TRUE' }
VERSION : 0.1
   VAR_TEMP
      size_before : Int;
      size_after : Int;
   END_VAR
BEGIN

   "fill_priority_queue"();

   IF "pq_is_empty"("DB_process_data".glass_queue) = FALSE
   THEN
       "DB_process_data".glass_queue.queue_array[0].glass.vehicle_model := 'IDBuzz';

       #size_before := "pq_size"("DB_process_data".glass_queue);

       IF "pq_dequeue"("DB_process_data".glass_queue) = true
       THEN
           #size_after := "pq_size"("DB_process_data".glass_queue);

           IF #size_before = #size_after + 1
               AND "DB_process_data".glass_queue.queue_array[0].glass.vehicle_model = 'T7'
           THEN
               #pq_dequeue_test := true;
           ELSE
               #pq_dequeue_test := false;
           END_IF;
       ELSE
           #pq_dequeue_test := false;
       END_IF;

       "pq_clear"("DB_process_data".glass_queue);
   ELSE
       #pq_dequeue_test := false;
   END_IF;
END_FUNCTION

FUNCTION "pq_peek_test" : Bool   // FC21, SCL
{ S7_Optimized_Access := 'TRUE' }
VERSION : 0.1
   VAR_TEMP
      node1 : "QueueNode";
      node2 : "QueueNode";
   END_VAR
BEGIN


   "fill_priority_queue"();

   IF "pq_is_empty"("DB_process_data".glass_queue) = FALSE
   THEN
       "DB_process_data".glass_queue.queue_array[5].glass.vehicle_model := 'IDBuzz';

       #node1 := "pq_peek"(index := 5, self := "DB_process_data".glass_queue);
       #node2 := "pq_peek"(index := 55, self := "DB_process_data".glass_queue);

       IF #node1.glass.vehicle_model = 'IDBuzz'
           AND #node2.glass.vehicle_model = ''
           AND #node2.glass.vehicle_number = ''
           AND #node2.glass.rear_window = ''
       THEN
           #pq_peek_test := true;
       ELSE
           #pq_peek_test := false;
       END_IF;

       "pq_clear"("DB_process_data".glass_queue);
   ELSE
       #pq_peek_test := false;
   END_IF;
END_FUNCTION

FUNCTION "pq_delete_by_index_test" : Bool   // FC22, SCL
{ S7_Optimized_Access := 'TRUE' }
VERSION : 0.1
   VAR_TEMP
      size_before : Int;
      size_after : Int;
   END_VAR
   VAR CONSTANT
      check_array_index : Int := 5;
   END_VAR
BEGIN


   "fill_priority_queue"();

   IF "pq_is_empty"("DB_process_data".glass_queue) = FALSE
   THEN
       "DB_process_data".glass_queue.queue_array[#check_array_index].glass.vehicle_model := 'IDBuzz';

       #size_before := "pq_size"("DB_process_data".glass_queue);

       IF "pq_delete_by_index"(index := #check_array_index, self := "DB_process_data".glass_queue) = TRUE
       THEN
           #size_after := "pq_size"("DB_process_data".glass_queue);

           IF #size_before = #size_after + 1
               AND "DB_process_data".glass_queue.queue_array[#check_array_index].glass.vehicle_model = 'T7'
           THEN
               #pq_delete_by_index_test := true;
           ELSE
               #pq_delete_by_index_test := false;
           END_IF;
       ELSE
           #pq_delete_by_index_test := false;
       END_IF;

       "pq_clear"("DB_process_data".glass_queue);
   ELSE
       #pq_delete_by_index_test := false;
   END_IF;
END_FUNCTION

FUNCTION "pq_is_empty_test" : Bool   // FC23, SCL
{ S7_Optimized_Access := 'TRUE' }
VERSION : 0.1
BEGIN


   IF "pq_is_empty"("DB_process_data".glass_queue) = TRUE
   THEN
       "fill_priority_queue"();

       IF "pq_is_empty"("DB_process_data".glass_queue) = FALSE
           AND "pq_size"("DB_process_data".glass_queue) > 0
       THEN
           #pq_is_empty_test := true;
       ELSE
           #pq_is_empty_test := false;
       END_IF;

       "pq_clear"("DB_process_data".glass_queue);
   ELSE
       #pq_is_empty_test := false;
   END_IF;
END_FUNCTION

FUNCTION "pq_size_test" : Bool   // FC24, SCL
{ S7_Optimized_Access := 'TRUE' }
VERSION : 0.1
   VAR_TEMP
      size_before : Int;
      size_after : Int;
   END_VAR
BEGIN

   IF "pq_is_empty"("DB_process_data".glass_queue) = TRUE
   THEN
       #size_before := "pq_size"("DB_process_data".glass_queue);
       "fill_priority_queue"();
       #size_after := "pq_size"("DB_process_data".glass_queue);

       IF "pq_is_empty"("DB_process_data".glass_queue) = FALSE
       THEN
           IF #size_before = 0
               AND #size_after = 50
           THEN
               #pq_size_test := true;
           ELSE
               #pq_size_test := false;
           END_IF;
       ELSE
           #pq_size_test := false;
       END_IF;

       "pq_clear"("DB_process_data".glass_queue);
   ELSE
       #pq_size_test := false;
   END_IF;
END_FUNCTION

FUNCTION "pq_find_by_vehicle_number_test" : Bool   // FC26, SCL
{ S7_Optimized_Access := 'TRUE' }
VERSION : 0.1
   VAR_TEMP
      glass1 : "GlassInfo";
      glass2 : "GlassInfo";
      glass3 : "GlassInfo";
   END_VAR
BEGIN

   IF "pq_is_empty"("DB_process_data".glass_queue) = TRUE
   THEN

       #glass1 := "gi_new"(rear_window := 'VW-0001', vehicle_model := 'T7',vehicle_number := '123456789 00');
       #glass2 := "gi_new"(rear_window := 'VW-0001', vehicle_model := 'T7', vehicle_number := '123456790 00');
       #glass3 := "gi_new"(rear_window := 'VW-0001', vehicle_model := 'T7', vehicle_number := '123456791 00');

       IF "pq_enqueue"(glass := #glass1, priority := false, self := "DB_process_data".glass_queue) = true
           AND "pq_enqueue"(glass := #glass2, priority := false, self := "DB_process_data".glass_queue) = true
           AND "pq_enqueue"(glass := #glass3, priority := false, self := "DB_process_data".glass_queue) = true
       THEN
           IF "pq_find_by_vehicle_number"(vehicle_number := '123456790 00', self := "DB_process_data".glass_queue) = 1
               AND "pq_find_by_vehicle_number"(vehicle_number := '123456790 01', self := "DB_process_data".glass_queue) = 1
           THEN
               #pq_find_by_vehicle_number_test := true;
           ELSE
               #pq_find_by_vehicle_number_test := false;
           END_IF;

           "pq_clear"("DB_process_data".glass_queue);
       ELSE
           #pq_find_by_vehicle_number_test := false;
       END_IF;
   ELSE
       #pq_find_by_vehicle_number_test := false;
   END_IF;
END_FUNCTION

// folder: unitLib/test_suites/priority_queue_test/pq_test_util

FUNCTION "fill_priority_queue" : Void   // FC28, SCL
{ S7_Optimized_Access := 'TRUE' }
VERSION : 0.1
   VAR_TEMP
      i : Int;
      glass : "GlassInfo";
      vehicle_number : String;
   END_VAR
BEGIN






   WHILE #i < 50 DO
       #vehicle_number := CONCAT(IN1 := INT_TO_STRING(#i), IN2 := ' 00');

       #glass := "gi_new"(rear_window := 'VW-Number', vehicle_model := 'T7', vehicle_number := #vehicle_number);

       IF "pq_enqueue"(glass := #glass, priority := false, self := "DB_process_data".glass_queue) = TRUE
       THEN
           #i := #i + 1;
       ELSE
           #i := "DB_process_data".glass_queue.array_size;
       END_IF;
   END_WHILE;
END_FUNCTION

(* ===== HMI "HMI_RT_1" =====
system functions are stored by id; their names below are inferred from use
connection "HMI_Connection_1": ETHERNET, SMART_S7_1200_OMS

HMI tags "Default tag table"
   "Valves_DB_test_valve_stat_error" : Bool = PLC Valves_DB.test_valve.status_error, 1 s
   "Valves_DB_test_valve_start_position_signal" : Bool = PLC Valves_DB.test_valve.cmd_start_position, 1 s
   "Valves_DB_test_valve_i_start_position" : Bool = PLC Valves_DB.test_valve.i_start_position, 1 s
   "Valves_DB_test_valve_i_end_position" : Bool = PLC Valves_DB.test_valve.i_end_position, 1 s
   "Valves_DB_test_valve_end_position_signal" : Bool = PLC Valves_DB.test_valve.cmd_end_position, 1 s
   "Valves_DB_test_valve_req_signal_start" : Bool = PLC Valves_DB.test_valve.request_signal_start, 1 s
   "Valves_DB_test_valve_req_signal_end" : Bool = PLC Valves_DB.test_valve.request_signal_end, 1 s
   "Valves_DB_test_valve_req_release" : Bool = PLC Valves_DB.test_valve.request_release, 1 s
   "i_test_vavlve_end" : Bool = PLC i_test_vavlve_end AT %M0.3, 1 s
   "i_test_valve_start" : Bool = PLC i_test_valve_start AT %M0.2, 1 s

screen "Screen_1" 800x480
   Button "Button_1" at 210,154 size 96x32; TextOff 'Start'
      on Press: function_b14e0dd5("Valves_DB_test_valve_req_signal_start", 0)
   Button "Button_2" at 489,155 size 96x32; TextOff 'End'
      on Press: function_b14e0dd5("Valves_DB_test_valve_req_signal_end", 0)
   Rectangle "Rectangle_1" at 210,131 size 376x16
      Appearance <- "Valves_DB_test_valve_stat_error"
   Rectangle "Rectangle_2" at 311,155 size 42x12
      Appearance <- "Valves_DB_test_valve_start_position_signal"
   Rectangle "Rectangle_3" at 311,175 size 42x12
      Appearance <- "Valves_DB_test_valve_i_start_position"
   Rectangle "Rectangle_4" at 441,155 size 42x12
      Appearance <- "Valves_DB_test_valve_end_position_signal"
   Rectangle "Rectangle_5" at 441,175 size 42x12
      Appearance <- "Valves_DB_test_valve_i_end_position"
   Switch "Switch_1" at 340,217 size 121x44; CaptionText 'Switch'; TextOff 'Release'; TextOn 'Release'
      ProcessValue <- "Valves_DB_test_valve_req_release"
      Appearance <- "Valves_DB_test_valve_req_release"
   Switch "Switch_2" at 520,71 size 64x32; CaptionText 'Switch'; TextOff 'OFF'; TextOn 'ON'
      ProcessValue <- "i_test_vavlve_end"
   Switch "Switch_3" at 210,71 size 64x32; CaptionText 'Switch'; TextOff 'OFF'; TextOn 'ON'
      ProcessValue <- "i_test_valve_start"
*)